// Restart after complete run
IF NOT Start_old AND Start THEN
	Index := 0;
	Finished := FALSE;
END_IF


CASE Index OF	
	0: // Switch to state 'Switch on disabled'
		IF (Start) THEN
			Mode_of_operation := E_Mode_of_operation.No_mode_active;
			Controlword := CONTROLWORD_STATE_CHANGE(Current_State, E_Statemachine_State.Switch_on_disabled);
			IF (Current_State = E_Statemachine_State.Switch_on_disabled) THEN			
				Index := Index + 2;
			ELSE
				Index := Index + 1;		
			END_IF
		END_IF
		
			
	1: // Wait for 'Switch on disabled'
		Controlword := CONTROLWORD_STATE_CHANGE(Current_State, E_Statemachine_State.Switch_on_disabled);	
		IF (Current_State = E_Statemachine_State.Switch_on_disabled) THEN			
			Index := Index + 1;		
		END_IF
					
		
	2: // Set Mode of operation
		Mode_of_operation := E_Mode_of_operation.Homing_mode;	
		Controlword := CONTROLWORD_STATE_CHANGE(Current_State, E_Statemachine_State.Switch_on_disabled);				
		IF (PDO.Mode_of_operation_display = E_Mode_of_operation.Homing_mode) THEN			
			IF Homing_parameters.Homing_mode = E_Homing_mode.Homing_on_current_position THEN
				Index := Index + 1 + 3*2;
			ELSE
				Index := Index + 1;		
			END_IF
		END_IF

		
	3: // Set Speed during search for switch		
		Controlword := CONTROLWORD_STATE_CHANGE(Current_State, E_Statemachine_State.Switch_on_disabled);	
		WriteData[0] := DWORD_TO_BYTE(Homing_parameters.Speed_switch);
		WriteData[1] := DWORD_TO_BYTE(SHR(Homing_parameters.Speed_switch,8));
		WriteData[2] := DWORD_TO_BYTE(SHR(Homing_parameters.Speed_switch,16));
		WriteData[3] := DWORD_TO_BYTE(SHR(Homing_parameters.Speed_switch,24));	
		SDO_WRITE(	
			AdsNetID		:= GLB.ADSNetID_CAN,
			PortNr			:= 16#1000 + GLB.NodeID,
			CO_Index		:= 16#6099,
			CO_SubIndex		:= 16#01,
			DataLength		:= 4,
			WriteData		:= WriteData,
			StartWriting	:= TRUE	
		);	
		Index := Index + 1;		
		
	4: // Wait for finish sdo transfer	
		Controlword := CONTROLWORD_STATE_CHANGE(Current_State, E_Statemachine_State.Switch_on_disabled);	
		SDO_WRITE(StartWriting := FALSE);
		IF SDO_WRITE.WriteDataFinished THEN
			Index := Index + 1;			
		END_IF	
		
		
	5: // Set Spped during search for zero			
		Controlword := CONTROLWORD_STATE_CHANGE(Current_State, E_Statemachine_State.Switch_on_disabled);	
		WriteData[0] := DWORD_TO_BYTE(Homing_parameters.Speed_zero);
		WriteData[1] := DWORD_TO_BYTE(SHR(Homing_parameters.Speed_zero,8));
		WriteData[2] := DWORD_TO_BYTE(SHR(Homing_parameters.Speed_zero,16));
		WriteData[3] := DWORD_TO_BYTE(SHR(Homing_parameters.Speed_zero,24));	
		SDO_WRITE(	
			AdsNetID		:= GLB.ADSNetID_CAN,
			PortNr			:= 16#1000 + GLB.NodeID,
			CO_Index		:= 16#6099,
			CO_SubIndex		:= 16#02,
			DataLength		:= 4,
			WriteData		:= WriteData,
			StartWriting	:= TRUE	
		);	
		Index := Index + 1;		
		
	6: // Wait for finish sdo transfer	
		Controlword := CONTROLWORD_STATE_CHANGE(Current_State, E_Statemachine_State.Switch_on_disabled);	
		SDO_WRITE(StartWriting := FALSE);
		IF SDO_WRITE.WriteDataFinished THEN
			Index := Index + 1;			
		END_IF		
		
		
	7: // Set Homing acceleration		
		Controlword := CONTROLWORD_STATE_CHANGE(Current_State, E_Statemachine_State.Switch_on_disabled);	
		WriteData[0] := DWORD_TO_BYTE(Homing_parameters.Acceleration);
		WriteData[1] := DWORD_TO_BYTE(SHR(Homing_parameters.Acceleration,8));
		WriteData[2] := DWORD_TO_BYTE(SHR(Homing_parameters.Acceleration,16));
		WriteData[3] := DWORD_TO_BYTE(SHR(Homing_parameters.Acceleration,24));	
		SDO_WRITE(	
			AdsNetID		:= GLB.ADSNetID_CAN,
			PortNr			:= 16#1000 + GLB.NodeID,
			CO_Index		:= 16#609A,
			CO_SubIndex		:= 16#00,
			DataLength		:= 4,
			WriteData		:= WriteData,
			StartWriting	:= TRUE	
		);	
		Index := Index + 1;		
		
	8: // Wait for finish sdo transfer	
		Controlword := CONTROLWORD_STATE_CHANGE(Current_State, E_Statemachine_State.Switch_on_disabled);	
		SDO_WRITE(StartWriting := FALSE);
		IF SDO_WRITE.WriteDataFinished THEN
			Index := Index + 1;			
		END_IF	
		
		
	9: // Set Homing mode		
		Controlword := CONTROLWORD_STATE_CHANGE(Current_State, E_Statemachine_State.Switch_on_disabled);	
		WriteData[0] := Homing_parameters.Homing_mode;
		SDO_WRITE(	
			AdsNetID		:= GLB.ADSNetID_CAN,
			PortNr			:= 16#1000 + GLB.NodeID,
			CO_Index		:= 16#6098,
			CO_SubIndex		:= 16#00,
			DataLength		:= 1,
			WriteData		:= WriteData,
			StartWriting	:= TRUE	
		);	
		Index := Index + 1;		
		
	10: // Wait for finish sdo transfer	
		Controlword := CONTROLWORD_STATE_CHANGE(Current_State, E_Statemachine_State.Switch_on_disabled);	
		SDO_WRITE(StartWriting := FALSE);
		IF SDO_WRITE.WriteDataFinished THEN
			Index := Index + 1;			
		END_IF		
		
		
	11: // Switch State to 'Operation enabled'
		Controlword := CONTROLWORD_STATE_CHANGE(Current_State, E_Statemachine_State.Operation_enabled);		
		IF (Current_State = E_Statemachine_State.Operation_enabled) THEN			
			Index := Index + 1;
		END_IF
		
		
	12: // Start homing and wait for finish
		Controlword := 16#1F;		
		IF (Statusword AND E_Statusword_Bits.HM_Homing_attained) <> 0 THEN			
			Index := Index + 1;		
		END_IF
	
		
	13: // Switch State to 'Switch on disabled'
		Controlword := CONTROLWORD_STATE_CHANGE(Current_State, E_Statemachine_State.Switch_on_disabled);	
		IF Current_State = E_Statemachine_State.Switch_on_disabled THEN			
			Index := 255;
		END_IF
		
		
	255: // Finished 
		Controlword := CONTROLWORD_STATE_CHANGE(Current_State, E_Statemachine_State.Switch_on_disabled);	
		FINISHED := TRUE;
				
		
	ELSE
		Index := 255;
			
END_CASE


Start_old := Start;

END_FUNCTION_BLOCK

// ---- POUs/FB/FB_Sequenz_Testing.TcPOU
FUNCTION_BLOCK FB_Sequenz_Testing
VAR_INPUT	
	Start			: BOOL 			:= FALSE;			// Start command
	Sequence_Name	: STRING(50) 	:= '';				// The name of the sequence
	Logging_active	: BOOL 			:= TRUE;			// The logging is default active. For deactivating set the variable to false.
END_VAR
VAR_OUTPUT
	Busy			: BOOL			:= FALSE;
	Finished		: BOOL			:= FALSE;			// The sequence is finished.
	Error			: BOOL			:= FALSE;			// Error during the sequence.
END_VAR
VAR_IN_OUT
	Step_list		: ARRAY [*] OF E_Test_step;	// Array with the sequence of steps
END_VAR
VAR
	Step_index		: DINT			:= 0;				// The current index of test step
	Step_state		: BYTE			:= 0;				// The internal state of the current test step
	Counter			: WORD			:= 0;				// Counter variable for internal use
	
	Name			: STRING(50)	:= '';				// The current sequence name. The name is saved once by start of the sequence.
	
	Data			: ARRAY [0..255] OF BYTE;
	CAN_Object		: ST_CAN_Object;	
	SDO_READ		: FB_SDO_READ;
	SDO_WRITE		: FB_SDO_WRITE;
	Write_busy		: BOOL 			:= FALSE;			// A writing process is running. After finishing the process the next test step is started
	Write_sequence	: BOOL			:= FALSE;			// If this Flag is set, the internal step state is increased. Otherwise the test step is finished after the write process.
	
	Next_Step_state	: BOOL 			:= FALSE;			// Increase the internal state of the test step
	Step_Finished	: BOOL 			:= FALSE;			// Switch to the next test step
	Error_step		: DINT 			:= -1;				// List index of the test state, at which an error is occured
	
	Current_Statemachine_state: E_Statemachine_State;	// The current State machine state
	
	Timeout_Counter	: INT			:= 0;				// Timeout Counter
	Timeout_Max		: INT			:= 0;				// Value at which the timeout counter is triggered (x 10 ms)

	Wait_Counter	: INT			:= 0;				// Wait Counter
	Wait_Step_Finish: BOOL			:= TRUE;			// True: The step is finished after the waiting time. False: The status counter in the step is increased after the waiting time.
	Wait_Time		: INT			:= 0;				// Value at which the wait counter is triggered (x 10 ms)

	Message			: STRING(60)	:= '';				// This message is send at the end of the FB
END_VAR

// Start / Reset
IF Start AND NOT Busy THEN
	Step_index		:= 0;
	Step_state 		:= 0;	
	Finished		:= FALSE;
	Error			:= FALSE;
	Error_step		:= -1;
 	Busy 			:= TRUE;	
	Name 			:= Sequence_Name;
	IF Sequence_Name = '' AND Logging_active THEN
		GLB.Logger(Message:='Start sequence');
	ELSE
		GLB.Logger(Message:=CONCAT('Start sequence: ', Sequence_Name)); 
	END_IF
END_IF


IF Busy THEN
	// Reached end?
	IF (Step_index > UPPER_BOUND(Step_list, 1)) OR (Error_step > -1) THEN
		Busy 		:= FALSE;
		Finished 	:= TRUE;
		IF Error_step = -1 AND Logging_active THEN
			GLB.Logger(Message:='Sequence successful', SaveFlag:=TRUE);
			Error	:= FALSE;
		ELSE	
			GLB.Logger(Message:='Sequence failed', SaveFlag:=TRUE);			
			Error	:= TRUE;		
		END_IF
				
	ELSE
		// Get the current state of the State machine
		Current_Statemachine_state 			:= GET_STATE(PDO.Statusword);
			
		// Processing the individual test steps  
		CASE Step_list[Step_index] OF
		
			// **** Change of state machine state *****
			// Switch directly to state 'Switch on disabled' -> Set Controlword to 0
			E_Test_step.Switch_on_disabled:
				CASE Step_state OF
					0:	// Set Controlword to 0
						PDO.Controlword			:= E_Statemachine_Transition_Controlword.Switch_on_disabled;
						Message					:= 'Switch to state Switch on disabled';		
						Next_Step_state			:= TRUE;
					
					1:	// Wait until state 'Switch on disabled'
						IF Current_Statemachine_state = E_Statemachine_State.Switch_on_disabled THEN		Step_Finished := TRUE;	END_IF	
				END_CASE	
				
			// Switch directly to state 'Quick stop active' -> Set Controlword to 2		
			E_Test_step.Quick_stop_active:
				CASE Step_state OF
					0:	// Set Controlword to 2
						PDO.Controlword			:= E_Statemachine_Transition_Controlword.Quick_stop_active;
						Message					:= 'Switch to state Quick stop active';		
						Next_Step_state			:= TRUE;
					
					1:	// Wait until state 'Quick stop active'
						IF Current_Statemachine_state = E_Statemachine_State.Quick_stop_active THEN			Step_Finished := TRUE;	END_IF
				END_CASE
													
			// Switch directly to state 'Ready to switch on' -> Set Controlword to 6		
			E_Test_step.Ready_to_switch_on:
				CASE Step_state OF
					0:	// Set Controlword to 6
						PDO.Controlword			:= E_Statemachine_Transition_Controlword.Ready_to_switch_on;
						Message					:= 'Switch to state Ready to switch on';			
						Next_Step_state			:= TRUE;				
				
					1:	// Wait until state 'Ready to switch on'
						IF Current_Statemachine_state = E_Statemachine_State.Ready_to_switch_on THEN		Step_Finished := TRUE;	END_IF
				END_CASE
													
			// Switch directly to state 'Switched on' -> Set Controlword to 7			
			E_Test_step.Switched_on:				
				CASE Step_state OF
					0:	// Set Controlword to 7
						PDO.Controlword			:= E_Statemachine_Transition_Controlword.Switched_on;
						Message					:= 'Switch to state Switched on';				
						Next_Step_state			:= TRUE;
					
					1:	// Wait until state 'Switched on'
						IF Current_Statemachine_state = E_Statemachine_State.Switched_on THEN				Step_Finished := TRUE;	END_IF
				END_CASE
													
			// Switch directly to state 'Operation enabled' -> Set Controlword to F		
			E_Test_step.Operation_enabled:				
				CASE Step_state OF
					0:	// Set Controlword to F
						PDO.Controlword			:= E_Statemachine_Transition_Controlword.Operation_enabled;
						Message					:= 'Switch to state Operation enabled';			
						Next_Step_state			:= TRUE;
					
					1:	// Wait until state 'Operation enabled'
						IF Current_Statemachine_state = E_Statemachine_State.Operation_enabled THEN			Step_Finished := TRUE;	END_IF
				END_CASE													
			// ****************************************	
						
			// ***** Change of Mode of Operation ******
			// Set Mode of Operation to 'No mode'
			E_Test_step.No_Mode:
				CASE Step_state OF
					0:
						PDO.Mode_of_operation	:= E_Mode_of_Operation.No_mode_active;
						Message					:= 'Set Mode of Operation to "No mode"';		
						Next_Step_state			:= TRUE;
					
					1:	// Wait until mode 'No mode'
						IF PDO.Mode_of_operation_display = E_Mode_of_Operation.No_mode_active THEN			Step_Finished := TRUE;	END_IF				
				END_CASE
						
			// Set Mode of Operation to 'Profile Position Mode'
			E_Test_step.Mode_PPM:
				CASE Step_state OF
					0:	
						PDO.Mode_of_operation	:= E_Mode_of_Operation.Profile_position_mode;
						Message					:= 'Set Mode of Operation to "Profile Position Mode"';			
						Next_Step_state			:= TRUE;
					
					1:	// Wait until mode 'Profile Position Mode'
						IF PDO.Mode_of_operation_display = E_Mode_of_Operation.Profile_position_mode THEN	Step_Finished := TRUE;	END_IF				
				END_CASE
								
			// Set Mode of Operation to 'Velocity Mode'
			E_Test_step.Mode_VM:
				CASE Step_state OF
					0:
						PDO.Mode_of_operation	:= E_Mode_of_Operation.Velocity_mode;
						Message					:= 'Set Mode of Operation to "Velocity Mode"';			
						Next_Step_state			:= TRUE;
					
					1:	// Wait until mode 'Velocity Mode'
						IF PDO.Mode_of_operation_display = E_Mode_of_Operation.Velocity_mode THEN			Step_Finished := TRUE;	END_IF		
				END_CASE
			
			// Set Mode of Operation to 'Profile Velocity Mode'
			E_Test_step.Mode_PVM:
				CASE Step_state OF
					0:
						PDO.Mode_of_operation	:= E_Mode_of_Operation.Profile_velocity_mode;
						Message					:= 'Set Mode of Operation to "Profile Velocity Mode"';			
						Next_Step_state			:= TRUE;
					
					1:	// Wait until mode 'Profile Velocity Mode'
						IF PDO.Mode_of_operation_display = E_Mode_of_Operation.Profile_velocity_mode THEN	Step_Finished := TRUE;	END_IF		
				END_CASE
										
			// Set Mode of Operation to 'Profile Torque Mode'
			E_Test_step.Mode_PTM:
				CASE Step_state OF
					0:
						PDO.Mode_of_operation	:= E_Mode_of_Operation.Profile_torque_mode;
						Message					:= 'Set Mode of Operation to "Profile Torque Mode"';		
						Next_Step_state			:= TRUE;
					
					1:	// Wait until mode 'Profile Torque Mode'
						IF PDO.Mode_of_operation_display = E_Mode_of_Operation.Profile_torque_mode THEN		Step_Finished := TRUE;	END_IF		
				END_CASE
				
			// Set Mode of Operation to 'Homing Mode'
			E_Test_step.Mode_HM:
				CASE Step_state OF
					0:
						PDO.Mode_of_operation	:= E_Mode_of_Operation.Homing_mode;
						Message					:= 'Set Mode of Operation to "Homing mode"';
						Next_Step_state			:= TRUE;
					
					1:	// Wait until mode 'Homing Mode'
						IF PDO.Mode_of_operation_display = E_Mode_of_Operation.Homing_mode THEN				Step_Finished := TRUE;	END_IF		
				END_CASE
										
			// Set Mode of Operation to 'Interpolated Position Mode'
			E_Test_step.Mode_IPM:
				CASE Step_state OF
					0:
						PDO.Mode_of_operation	:= E_Mode_of_Operation.Interpolated_position_mode;
						Message					:= 'Set Mode of Operation to "Interpolated Position Mode"';
						Next_Step_state			:= TRUE;
					
					1:	// Wait until mode 'Interpolated Position Mode'
						IF PDO.Mode_of_operation_display = E_Mode_of_Operation.Interpolated_position_mode THEN	Step_Finished := TRUE;	END_IF		
				END_CASE
			// ****************************************	
						
			// ************** Init steps **************	
			// Set the factor group to use rpm as user-defined velocity unit
			E_Test_step.Factor_group_rpm:
				Write_busy := TRUE;
				CASE Step_state OF
					0:	// Set ...
						Write_sequence := TRUE;
						DWORD_TO_BYTE_ARRAY(4096, Data);			
						CAN_Object 		:= DS402_Object_List.Velocity_Factor_Numerator;
						
					2:	// Set ...
						Write_sequence := FALSE;					
						DWORD_TO_BYTE_ARRAY(60, Data);			
						CAN_Object 		:= DS402_Object_List.Velocity_Factor_Divisor;
						
						
						
				END_CASE	
			// ****************************************	
			
			// ************ Setting values ************	
			// Set 'Velocity_window' to value 30
			E_Test_step.Velocity_window_30rpm:
				CASE Step_state OF
					0:
						DWORD_TO_BYTE_ARRAY(30, Data);			
						CAN_Object 		:= DS402_Object_List.Velocity_window;
						Message 		:= 'Set Velocity_window to 30';					
						Write_busy		:= TRUE;		
				END_CASE
			
			// Set 'Velocity window time' to value 100
			E_Test_step.Velocity_window_100ms:
				CASE Step_state OF
					0:
						DWORD_TO_BYTE_ARRAY(100, Data);			
						CAN_Object 		:= DS402_Object_List.Velocity_window_time;
						Message			:= 'Set Velocity window time to 100';					
						Write_busy		:= TRUE;
				END_CASE
				
			// Set 'Profile acceleration' to value 1000
			E_Test_step.Acceleration_1000:
				CASE Step_state OF
					0:
						DWORD_TO_BYTE_ARRAY(1000, Data);			
						CAN_Object 		:= DS402_Object_List.Profile_acceleration;
						Message			:= 'Set Profile acceleration to 1000';
						Write_busy		:= TRUE;	
				END_CASE
				
			// Set 'Profile deceleration' to value 1000			
			E_Test_step.Deceleration_1000:
				CASE Step_state OF
					0:
						DWORD_TO_BYTE_ARRAY(1000, Data);	
						CAN_Object 		:= DS402_Object_List.Profile_deceleration; 				
						Message			:= 'Set Profile deceleration to 1000';
						Write_busy		:= TRUE;
				END_CASE
				
			// Set 'Profile velocity' to value 1000			
			E_Test_step.PPM_Velocity_1000:
				CASE Step_state OF
					0:
						DWORD_TO_BYTE_ARRAY(1000, Data);			
						CAN_Object 		:= DS402_Object_List.Profile_velocity;
						Message			:= 'Set Profile velocity to 1000';					
						Write_busy		:= TRUE;	
				END_CASE
	
			// Set 'Target velocity' to value 1000
			E_Test_step.PVM_Velocity_1000:
				CASE Step_state OF
					0:	
						DWORD_TO_BYTE_ARRAY(1000, Data);			
						CAN_Object 		:= DS402_Object_List.Target_velocity;
						Message			:= 'Set Target velocity to 1000';
						Write_busy		:= TRUE;
				END_CASE		
			// ****************************************	
							
			// *********** Check conditions ***********
			// Check if the 'Target reached' bit in statusword is set within 200 ms
			E_Test_step.Check_Statusword_Target_reached_200ms:
				Timeout_Max 		:= 20;
				IF (PDO.Statusword AND E_Statusword_Bits.Target_reached) = E_Statusword_Bits.Target_reached THEN
					Message			:= 'Target reached bit is set';
					Step_Finished	:= TRUE;					
				END_IF	
			// ****************************************				
			
			// ************ Waiting times *************
			E_Test_step.Wait_10ms:		IF Step_state = 0 THEN	Wait_Time := 1; 	Message := 'Wait Time 10 ms is running';	Next_Step_State:=TRUE; END_IF
			E_Test_step.Wait_50ms:		IF Step_state = 0 THEN	Wait_Time := 5; 	Message := 'Wait Time 50 ms is running';	Next_Step_State:=TRUE; END_IF
			E_Test_step.Wait_100ms:		IF Step_state = 0 THEN	Wait_Time := 10; 	Message := 'Wait Time 100 ms is running';	Next_Step_State:=TRUE; END_IF
			E_Test_step.Wait_250ms:		IF Step_state = 0 THEN	Wait_Time := 25; 	Message := 'Wait Time 250 ms is running';	Next_Step_State:=TRUE; END_IF
			E_Test_step.Wait_500ms:		IF Step_state = 0 THEN	Wait_Time := 50; 	Message := 'Wait Time 500 ms is running';	Next_Step_State:=TRUE; END_IF
			E_Test_step.Wait_1000ms:	IF Step_state = 0 THEN	Wait_Time := 100; 	Message := 'Wait Time 1 s is running';		Next_Step_State:=TRUE; END_IF
			E_Test_step.Wait_2500ms:	IF Step_state = 0 THEN	Wait_Time := 250; 	Message := 'Wait Time 2.5 s is running';	Next_Step_State:=TRUE; END_IF
			// Feel free to create your own needed wait times :-)
			// ****************************************		
						
			ELSE
				// unknown steps -> next step
				Message				:= CONCAT(CONCAT('FB_Start_Testing: ERROR, unknown test step (', DINT_TO_STRING(Step_index)), ')');
				Step_Finished		:= TRUE;
	
		END_CASE
		
		// Waiting time. Active, if Wait_Time is greater than 0
		IF Wait_Time > 0 THEN
			Wait_Counter			:= Wait_Counter + 1;	
			IF Wait_Counter >= Wait_Time THEN
				Message				:= 'Waiting time expired';			
				IF Wait_Step_Finish THEN 
					Step_Finished	:= TRUE;
				ELSE
					Next_Step_state	:= TRUE;
				END_IF
			END_IF
		END_IF
		
		// SDO Write process is running. This generell function is used, if Write_busy is set.
		IF Write_busy THEN
			IF Step_state.0 = 0 THEN
				// Start writing
				SDO_Write(
					ADSNetID		:= GLB.ADSNetID_CAN,				
					PortNr 		 	:= 16#1000 + GLB.NodeID,
					CO_Index 		:= CAN_Object.Index,
					CO_SubIndex 	:= CAN_Object.Subindex,
					DataLength 		:= CAN_Object.Length,
					WriteData		:= Data,
					StartWriting	:= TRUE	);
				Next_Step_state	:= TRUE;								
			ELSE
				// Wait for finishing
				SDO_Write(StartWriting:=FALSE);
				IF SDO_WRITE.WriteDataFinished THEN
					Write_busy			:= FALSE;
					IF SDO_WRITE.Error = 0 THEN									
						IF Write_sequence THEN
							Next_step_state	:= TRUE;
						ELSE						
							Step_Finished	:= TRUE;
						END_IF;
					ELSE
						Message			:= CONCAT('ERROR: Write failed, Errornumber: ', DWORD_TO_HEXSTR(SDO_WRITE.Error, 8, FALSE));
						Error_step		:= Step_index;		
					END_IF	
					SDO_Write();	
				END_IF
			END_IF
		END_IF
		
		// Next Test step
		IF Step_Finished THEN
			IF Message = '' THEN Message := 'OK'; END_IF
			Step_Finished 			:= FALSE;
			Step_index				:= Step_index + 1;
			Step_state 				:= 0;
			Wait_Counter			:= 0;
			Wait_Time				:= 0;
			Wait_Step_Finish		:= TRUE;
			Write_sequence			:= FALSE;
			Timeout_Counter			:= 0;
			Timeout_Max 			:= 10;			// Set Timeout to a default value of 10 (= 100 ms)
			
		// Next internal state of the test step			
		ELSIF Next_Step_state THEN
			Next_Step_state			:= FALSE;
			Step_state				:= Step_state + 1;
			Timeout_Counter			:= 0;	
		
		// Timeout
		ELSE
			IF Timeout_Max > 0 THEN
				IF Timeout_Counter >= Timeout_Max THEN
					Message			:= CONCAT(CONCAT('Timeout triggered (', INT_TO_STRING(Timeout_Max * 10)), ' ms)');
					Error_step		:= Step_index;
				END_IF
				Timeout_Counter	:= Timeout_Counter + 1;	
			END_IF
		END_IF
	END_IF
	
	
	// Log message
	IF Message <> '' AND Logging_active  THEN
		GLB.Logger(Message:=Message);
		Message := '';
	END_IF
END_IF

END_FUNCTION_BLOCK

// ---- POUs/GET_STATE.TcPOU
FUNCTION GET_STATE : E_Statemachine_State
VAR_INPUT
	Statusword: WORD;
END_VAR
VAR_OUTPUT
	State : E_Statemachine_State;
END_VAR
VAR_STAT
	State_State: ARRAY[0..7] OF E_Statemachine_State := [
		E_Statemachine_State.Not_ready_to_switch_on,
		E_Statemachine_State.Switch_on_disabled,
		E_Statemachine_State.Ready_to_switch_on,
		E_Statemachine_State.Switched_on,
		E_Statemachine_State.Operation_enabled,
		E_Statemachine_State.Quick_stop_active,
		E_Statemachine_State.Fault_reaction_active,
		E_Statemachine_State.Fault];
			
	State_Statusword: ARRAY[0..7] OF WORD := [ 
		16#00,	// Not ready to switch on
		16#40, 	// Switch on disabled
		16#21, 	// Ready to switch on
		16#23, 	// Switched on
		16#27, 	// Operation enable
		16#07, 	// Quick_stop_active
		16#0F,	// Fault_reaction_active
		16#08];	// Fault
		
	State_Mask: ARRAY[0..7] OF WORD := [ 
		16#4F,	// Not ready to switch on
		16#4F, 	// Switch on disabled
		16#6F, 	// Ready to switch on
		16#6F, 	// Switched on
		16#6F, 	// Operation enable
		16#6F, 	// Quick_stop_active
		16#4F,	// Fault_reaction_active
		16#4F];	// Fault	
END_VAR
VAR
	i: INT;
END_VAR

FOR i := 0 TO 7 DO
	IF (Statusword AND State_Mask[i]) = State_Statusword[i] THEN
		State 		:= State_State[i];
		GET_STATE 	:= State_State[i];
		EXIT;
	END_IF
END_FOR

END_FUNCTION

// ---- POUs/Velocity_Mode.TcPOU
FUNCTION_BLOCK Velocity_Mode
VAR_INPUT
	NodeID			: BYTE; (* This Port No. addresses the CANopen Node (see System Manager) *)
	Start 			: BOOL;
	Current_State 	: E_Statemachine_State;	
	Statusword		: WORD;	
	Velocity_parameters	: ST_Velocity_parameters;
END_VAR
VAR_OUTPUT
	Controlword 	: WORD;
	Mode_of_operation 	: E_Mode_of_operation	:= E_Mode_of_operation.No_mode_active;
	vl_target_velocity	: INT := 0;	
	Finished		: BOOL;
END_VAR
VAR
	Index 			: BYTE := 0;
	
	SDO_WRITE		: FB_SDO_WRITE;
	WriteData		: ARRAY [0..255] OF BYTE;
	
	SDO_READ		: FB_SDO_READ;
	ReadStart		: BOOL;
	ReadError		: DWORD;
	ReadData		: ARRAY [0..255] OF BYTE;
	
	fbTonDelay		: TON;
	Start_old		: BOOL := FALSE;
END_VAR

// Restart after complete run
IF NOT Start_old AND Start THEN
	Index := 0;
	Finished := FALSE;
END_IF


CASE Index OF	
	0: // Switch to state 'Switch on disabled'
		IF (Start) THEN
			Mode_of_operation := E_Mode_of_operation.No_mode_active;
			vl_target_velocity := 0;			
			Controlword := CONTROLWORD_STATE_CHANGE(Current_State, E_Statemachine_State.Switch_on_disabled);
			IF (Current_State = E_Statemachine_State.Switch_on_disabled) THEN			
				Index := Index + 2;
			ELSE
				Index := Index + 1;		
			END_IF
		END_IF
		
			
	1: // Wait for 'Switch on disabled'
		Controlword := CONTROLWORD_STATE_CHANGE(Current_State, E_Statemachine_State.Switch_on_disabled);	
		IF (Current_State = E_Statemachine_State.Switch_on_disabled) THEN			
			Index := Index + 1;		
		END_IF
					
		
	2: // Set Mode of operation and Acceleration
		Mode_of_operation := E_Mode_of_operation.Velocity_mode;	
		Controlword := CONTROLWORD_STATE_CHANGE(Current_State, E_Statemachine_State.Switch_on_disabled);				
		WriteData[0] := DWORD_TO_BYTE(Velocity_parameters.vl_velocity_acceleration);
		WriteData[1] := DWORD_TO_BYTE(SHR(Velocity_parameters.vl_velocity_acceleration,8));
		WriteData[2] := DWORD_TO_BYTE(SHR(Velocity_parameters.vl_velocity_acceleration,16));
		WriteData[3] := DWORD_TO_BYTE(SHR(Velocity_parameters.vl_velocity_acceleration,24));	
		SDO_WRITE(	
			AdsNetID		:= GLB.ADSNetID_CAN,
			PortNr			:= 16#1000 + GLB.NodeID,
			CO_Index		:= 16#6048,
			CO_SubIndex		:= 16#00,
			DataLength		:= 4,
			WriteData		:= WriteData,
			StartWriting	:= TRUE	
		);	
		Index := Index + 1;		
		
	3: // Wait for finish sdo transfer	
		Controlword := CONTROLWORD_STATE_CHANGE(Current_State, E_Statemachine_State.Switch_on_disabled);	
		SDO_WRITE(StartWriting := FALSE);
		IF SDO_WRITE.WriteDataFinished THEN
			Index := Index + 1;			
		END_IF	
		
		
	4: // Set Deceleration			
		Controlword := CONTROLWORD_STATE_CHANGE(Current_State, E_Statemachine_State.Switch_on_disabled);	
		WriteData[0] := DWORD_TO_BYTE(Velocity_parameters.vl_velocity_deceleration);
		WriteData[1] := DWORD_TO_BYTE(SHR(Velocity_parameters.vl_velocity_deceleration,8));
		WriteData[2] := DWORD_TO_BYTE(SHR(Velocity_parameters.vl_velocity_deceleration,16));
		WriteData[3] := DWORD_TO_BYTE(SHR(Velocity_parameters.vl_velocity_deceleration,24));	
		SDO_WRITE(	
			AdsNetID		:= GLB.ADSNetID_CAN,
			PortNr			:= 16#1000 + GLB.NodeID,
			CO_Index		:= 16#6049,
			CO_SubIndex		:= 16#00,
			DataLength		:= 4,
			WriteData		:= WriteData,
			StartWriting	:= TRUE	
		);	
		Index := Index + 1;		
		
	5: // Wait for finish sdo transfer	
		Controlword := CONTROLWORD_STATE_CHANGE(Current_State, E_Statemachine_State.Switch_on_disabled);	
		SDO_WRITE(StartWriting := FALSE);
		IF SDO_WRITE.WriteDataFinished THEN
			Index := Index + 1;			
		END_IF		
		
		
	6: // Set Velocity and switch State to 'Operation enabled'
		vl_target_velocity := Velocity_parameters.vl_target_velocity;
		Controlword := CONTROLWORD_STATE_CHANGE(Current_State, E_Statemachine_State.Operation_enabled);		
		IF (Current_State = E_Statemachine_State.Operation_enabled) THEN			
			Index := 255;
		END_IF
				
		
	255: // Finished 
		Controlword := CONTROLWORD_STATE_CHANGE(Current_State, E_Statemachine_State.Switch_on_disabled);	
		FINISHED := TRUE;
				
		
	ELSE
		Index := 255;
			
END_CASE


Start_old := Start;

END_FUNCTION_BLOCK

// ---- POUs/Profile_Velocity_Mode.TcPOU
FUNCTION_BLOCK Profile_Velocity_Mode
VAR_INPUT
	NodeID					: BYTE; (* This Port No. addresses the CANopen Node (see System Manager) *)
	Start 					: BOOL;
	Current_State 			: E_Statemachine_State;	
	Statusword				: WORD;	
	Profile_velocity_parameters	: ST_Profile_velocity_parameters;
END_VAR
VAR_OUTPUT
	Controlword 			: WORD;
	Mode_of_operation 		: E_Mode_of_operation	:= E_Mode_of_operation.No_mode_active;
	Target_velocity			: DINT;
	Encoder_offset			: WORD;
	Finished				: BOOL;
END_VAR
VAR
	Index 			: BYTE := 0;
	
	SDO_WRITE		: FB_SDO_WRITE;
	WriteData		: ARRAY [0..255] OF BYTE;
	
	Start_old		: BOOL := FALSE;
END_VAR

// Restart after complete run
IF NOT Start_old AND Start THEN
	Index := 0;
	Finished := FALSE;
END_IF


CASE Index OF	
	0: // Switch to state 'Switch on disabled'
		IF (Start) THEN
			Mode_of_operation := E_Mode_of_operation.No_mode_active;
			Target_velocity	:= 0;	
			Controlword := CONTROLWORD_STATE_CHANGE(Current_State, E_Statemachine_State.Switch_on_disabled);
			IF (Current_State = E_Statemachine_State.Switch_on_disabled) THEN			
				Index := Index + 2;
			ELSE
				Index := Index + 1;		
			END_IF
		END_IF
		
			
	1: // Wait for 'Switch on disabled'
		Controlword := CONTROLWORD_STATE_CHANGE(Current_State, E_Statemachine_State.Switch_on_disabled);	
		IF (Current_State = E_Statemachine_State.Switch_on_disabled) THEN			
			Index := Index + 1;		
		END_IF
		
		
	2: // Set Mode of operation and Acceleration
		Mode_of_operation := E_Mode_of_operation.Profile_velocity_mode;	
		Controlword := CONTROLWORD_STATE_CHANGE(Current_State, E_Statemachine_State.Switch_on_disabled);				
		WriteData[0] := DWORD_TO_BYTE(Profile_velocity_parameters.Profile_acceleration);
		WriteData[1] := DWORD_TO_BYTE(SHR(Profile_velocity_parameters.Profile_acceleration,8));
		WriteData[2] := DWORD_TO_BYTE(SHR(Profile_velocity_parameters.Profile_acceleration,16));
		WriteData[3] := DWORD_TO_BYTE(SHR(Profile_velocity_parameters.Profile_acceleration,24));	
		SDO_WRITE(	
			AdsNetID		:= GLB.ADSNetID_CAN,
			PortNr			:= 16#1000 + GLB.NodeID,
			CO_Index		:= 16#6083,
			CO_SubIndex		:= 16#00,
			DataLength		:= 4,
			WriteData		:= WriteData,
			StartWriting	:= TRUE	
		);	
		Index := Index + 1;		
		
	3: // Wait for finish sdo transfer	
		Controlword := CONTROLWORD_STATE_CHANGE(Current_State, E_Statemachine_State.Switch_on_disabled);	
		SDO_WRITE(StartWriting := FALSE);
		IF SDO_WRITE.WriteDataFinished THEN
			Index := Index + 1;			
		END_IF	
		
		
	4: // Set Deceleration			
		Controlword := CONTROLWORD_STATE_CHANGE(Current_State, E_Statemachine_State.Switch_on_disabled);	
		WriteData[0] := DWORD_TO_BYTE(Profile_velocity_parameters.Profile_deceleration);
		WriteData[1] := DWORD_TO_BYTE(SHR(Profile_velocity_parameters.Profile_deceleration,8));
		WriteData[2] := DWORD_TO_BYTE(SHR(Profile_velocity_parameters.Profile_deceleration,16));
		WriteData[3] := DWORD_TO_BYTE(SHR(Profile_velocity_parameters.Profile_deceleration,24));	
		SDO_WRITE(	
			AdsNetID		:= GLB.ADSNetID_CAN,
			PortNr			:= 16#1000 + GLB.NodeID,
			CO_Index		:= 16#6084,
			CO_SubIndex		:= 16#00,
			DataLength		:= 4,
			WriteData		:= WriteData,
			StartWriting	:= TRUE	
		);	
		Index := Index + 1;		
		
	5: // Wait for finish sdo transfer	
		Controlword := CONTROLWORD_STATE_CHANGE(Current_State, E_Statemachine_State.Switch_on_disabled);	
		SDO_WRITE(StartWriting := FALSE);
		IF SDO_WRITE.WriteDataFinished THEN
			Index := Index + 1;			
		END_IF					
		
	6: // Set  velocity	
		Controlword := CONTROLWORD_STATE_CHANGE(Current_State, E_Statemachine_State.Switch_on_disabled);	
		Target_velocity	:= Profile_velocity_parameters.Target_velocity;
		Index := Index + 1;		
		
	7: // Switch State to 'Operation enabled'
		Controlword := CONTROLWORD_STATE_CHANGE(Current_State, E_Statemachine_State.Operation_enabled);		
		IF (Current_State = E_Statemachine_State.Operation_enabled) THEN			
			Index := 255;
		END_IF
				
		
	255: // Finished 
		FINISHED := TRUE;
				
		
	ELSE
		Index := 255;
			
END_CASE


Start_old := Start;

END_FUNCTION_BLOCK

// ---- POUs/FUN/DWORD_TO_BYTE_ARRAY.TcPOU
FUNCTION DWORD_TO_BYTE_ARRAY
VAR_INPUT
	Value	: DWORD;
END_VAR
VAR_IN_OUT
	DATA	: ARRAY [*] OF BYTE;
END_VAR
VAR
	i		: BYTE := 0;
END_VAR

FOR i := 0 TO 3 DO
	DATA[i] := DWORD_TO_BYTE(SHR(Value, (8*i)));			
END_FOR;

END_FUNCTION

// ---- POUs/J_Stop_Testing_SM.TcPOU
FUNCTION_BLOCK J_Stop_Testing_SM
VAR_INPUT
	JST_NodeID					: BYTE; (* This Port No. addresses the CANopen Node (see System Manager) *)
	JST_Start_Testing			: BOOL; (* Send True to start the Stop Testing*)
	JST_Current_State 			: E_Statemachine_State;
END_VAR
VAR_OUTPUT
	Finished 					: BOOL := FALSE;
	JST_Controlword 			: WORD;
	Mode_of_operation 			: E_Mode_of_operation	:= E_Mode_of_operation.No_mode_active;
END_VAR
VAR
	// Statemachine variables
	e_Controlword_Send : (Wait_For_Send, Continue_SM) := Continue_SM;
	
	JST_Profile_Velocity_Mode 		: Profile_Velocity_Mode;
	e_Stop_Testing_State_Machine 	: (Idle,
									   Initialise_Drive,
									   Check_Start_Drive_Condition,
									   Change_Stop_Testing_State,
								       Stop_Testing, 
									   Check_Stop_Drive_Condition,
									   Start_Drive, 
									   Error_Handling); 
									
	e_Operation_Mode : E_Mode_of_operation := E_Mode_of_operation.Velocity_mode;
	
	(* e_Stop_Mode :  (Switch_On,					//schnell runterrampen -> Switched on
					Shutdown,					//Disable PS
					Switch_On_Disabled,			//Disable PS
					Vel_To_Zero,				//Ramp down
					Halt,						//stillstand mit dehmoment -> Weiterdrehen
					Quick_Stop,					//schnell runterrampen -> Switch on Disabled
					STO1,						//Disable PS
					STO2,						//Disable PS
					Fault						//DISABLE PS
					) := Switch_On; *)
	
	e_Stop_Mode : J_E_Stop_Modes := J_E_Stop_Modes.Switch_On;
	
	e_Stop_Type :  (Idle_Output_Stage,
				    Ramp_Down_AFAP,
					Vel_Zero);
					
	e_Start_Type : (Start_After_Reset,
					No_Start_After_Reset);
					
	
	JST_Profile_velocity_parameters	: ST_Profile_velocity_parameters := (Target_velocity 	  := 1000,
																 		 Profile_acceleration := 1000,
																 		 Profile_deceleration := 1000);
																 
	Target_velocity	: INT := 0;
	Target_State : E_STATEMACHINE_STATE;
	
	SDO_WRITE		: FB_SDO_WRITE;
	WriteData		: ARRAY [0..255] OF BYTE;
	
	//Tolerance variables
	Time_Tolerance : INT := 20;		//Unit is ms
	Vel_Tolerance  : INT := 30;		//Assumed that unit is RPM
	Stop_Tolerance : INT := 5;
	Stop_Time_AFAP : TIME := T#500MS;
	
	// Trash Variables 
	Temp 				         : BOOL := TRUE;
	JumpNextState 				 : BOOL := FALSE;
	Quick_Stop_Activ_Reset 		 : WORD := 16#00;
	Mode_Change 				 : BOOL := TRUE;
	Temp_msg 					 : STRING; 
	Delay 						 : BOOL := FALSE;
	Send_Controlword_Direct 	 : BOOL := FALSE;
	Quickstop_Change_Controlword : BOOL := TRUE;
	
	//Timer variables
	Toff : TIME := T#2000MS;
	
	StopTimer			 : TON := (PT := Toff);
	StartDelayTimer 	 : TON := (PT := Toff);
	CheckStartDelayTimer : TON := (PT := Toff);
	
	Stop_Timer 			: BOOL;
	Start_Delay_Timer 		: BOOL;
	Check_Start_Delay_Timer : BOOL;
	
	Elapsed_Time 			: TIME;
	
	//Message logging variables
	//fb_Message_Logging 		: J_Make_Message;
	Stop_Mode_String 		: STRING;
	
	// 24V Output variables
	OutputSTO1 	AT%Q* 		: BOOL;
	OutputSTO2 	AT%Q* 		: BOOL;

	Actual_Velocity_RPM		: DINT;
END_VAR

StopTimer(IN := Stop_Timer);
StartDelayTimer(IN := Start_Delay_Timer);
CheckStartDelayTimer(IN := Check_Start_Delay_Timer);

Actual_Velocity_RPM := PDO.vl_Velocity_actual_value;
//e_Operation_Mode := PDO.Mode_of_operation_display;

CASE e_Controlword_Send OF
	Continue_SM:		
		CASE e_Stop_Testing_State_Machine OF
			
			Idle:
				IF JST_Start_Testing THEN
					e_Stop_Testing_State_Machine := Initialise_Drive;
					e_Operation_Mode := E_Mode_of_operation.Velocity_mode;
					Finished := FALSE;
					GLB.Logger.OpenFlag := TRUE;
				ELSE
					e_Stop_Testing_State_Machine := Idle;
				END_IF
				
		//_____________________Start Drive SM___________________________________
			Initialise_Drive:
				OutputSTO1 := TRUE;
				OutputSTO2 := TRUE;
				CASE e_Operation_Mode OF
					//----------------------------------------------------------
					E_Mode_of_operation.Profile_position_mode:
						// Vel = 1000 ; Acc = 1000 ; Dec = 1000, Pos = 10000000						  
						IF NOT JST_Profile_Velocity_Mode.Finished THEN
							//just want to set acc and dec but not enable the drive
							JST_Profile_Velocity_Mode (NodeID := JST_NodeID,		//PVM just because the param for acc and dec are set and the same as in PPM
													   Start := TRUE,
													   Current_State := JST_Current_State,
													   Statusword := PDO.Statusword,
													   Profile_velocity_parameters := JST_Profile_velocity_parameters,
													   Controlword => JST_Controlword);
							e_Controlword_Send := Continue_SM;
							
						ELSIF JST_Profile_Velocity_Mode.Finished THEN

							PDO.Mode_of_operation 	:= E_Mode_of_operation.Profile_position_mode;		
							PDO.Profile_velocity 	:= JST_Profile_velocity_parameters.Target_velocity;
							PDO.Target_position 	:= 16#1000000;    // need to evaluate a good value 
							
							//Profile position FB how to use?
							Target_State := E_Statemachine_State.Operation_enabled;
							e_Controlword_Send := Wait_For_Send;
							e_Stop_Testing_State_Machine := Check_Start_Drive_Condition;
							Mode_Change := TRUE;
						END_IF
					//----------------------------------------------------------					
					E_Mode_of_operation.Velocity_mode:
							// Vel = 1000
							PDO.Mode_of_operation := E_Mode_of_Operation.Velocity_mode;
							PDO.vl_target_velocity := TO_INT(JST_Profile_velocity_parameters.Target_velocity);
							Target_State := E_Statemachine_State.Operation_enabled;
							e_Controlword_Send := Wait_For_Send;
							e_Stop_Testing_State_Machine := Check_Start_Drive_Condition;
							Check_Start_Delay_Timer := TRUE;	
		
					//----------------------------------------------------------	
					E_Mode_of_operation.Profile_velocity_mode:
						// Vel = 1000 ; Acc = 1000 ; Dec = 500
						// Start Drive, Wait for SDO written then change state
						IF NOT JST_Profile_Velocity_Mode.Finished THEN
							JST_Profile_Velocity_Mode (NodeID := JST_NodeID,
													   Start := TRUE,
													   Current_State := JST_Current_State,
													   Statusword := JST_Current_State,
													   Profile_velocity_parameters := JST_Profile_velocity_parameters,
													   Controlword => JST_Controlword);
							e_Controlword_Send := Continue_SM;
							
						ELSIF JST_Profile_Velocity_Mode.Finished THEN
							PDO.Profile_velocity := JST_Profile_velocity_parameters.Target_velocity;
							e_Stop_Testing_State_Machine := Check_Start_Drive_Condition;
						END_IF
					//----------------------------------------------------------
					E_Mode_of_operation.Profile_torque_mode:
						Target_State := E_Statemachine_State.Ready_to_switch_on;
						e_Controlword_Send := Wait_For_Send;
							IF PDO.Controlword = E_Statusword_Bits.Ready_to_switch_on THEN
								PDO.Mode_of_operation := E_Mode_of_Operation.Profile_torque_mode;
								PDO.Target_torque := 100; 	// Asssumed unit is in Promill
								Target_State := E_Statemachine_State.Operation_enabled;
								e_Controlword_Send := Wait_For_Send;
								e_Stop_Testing_State_Machine := Check_Start_Drive_Condition;
							END_IF	
				END_CASE
				e_Start_Type := Start_After_Reset;
				
		//__________________Check Drive Condition SM_____________________________
			Check_Start_Drive_Condition:
				// Wait for desired speed 
				IF CheckStartDelayTimer.Q THEN
					Check_Start_Delay_Timer := FALSE;  // Kann zu problemen führen, da falls der timer gleich resettet wird auch der programmzeiger nichtmehr in die If reinhüpft
					CASE e_Operation_Mode OF
						//-----------------------------------------------------------
						E_Mode_of_operation.Profile_position_mode, E_Mode_of_operation.Velocity_mode, E_Mode_of_operation.Profile_velocity_mode:
							CASE e_Start_Type OF
								Start_After_Reset:
									IF ABS(Actual_Velocity_RPM - JST_Profile_velocity_parameters.Target_velocity) < Vel_Tolerance THEN
									  // AND PDO.Statusword = E_Statusword_Bits.Target_reached THEN  //hier nochmal nachschauen
											// e_Stop_Mode muss mitgeloggt werden!!! sonst erkennt man nicht in welchem fall der motor wieder anläuft
											GLB.Logger.Message := J_Make_Message( Testing_Mode := e_Stop_Mode,
																					  Operation_Mode := e_Operation_Mode,
																				      Desired_Value := JST_Profile_velocity_parameters.Target_velocity,
																				      Real_Value := TO_INT(Actual_Velocity_RPM),
																				      Ranking := J_E_Test_Ranking.OK,
																				      Comment := 'Drive started in toleran'); 									   
											ADSLOGSTR(msgCtrlMask := ADSLOG_MSGTYPE_ERROR OR ADSLOG_MSGTYPE_LOG,
													msgFmtStr := CONCAT('Geschwindigkeit passt  ',TO_STRING(Actual_Velocity_RPM)),
													strArg := '');
											e_Stop_Testing_State_Machine := Change_Stop_Testing_State;
									
									ELSIF ABS(Actual_Velocity_RPM - JST_Profile_velocity_parameters.Target_velocity) < Vel_Tolerance THEN
										J_Make_Message(Testing_Mode := e_Stop_Mode,
														   Operation_Mode := e_Operation_Mode,
														   Desired_Value := JST_Profile_velocity_parameters.Target_velocity,
														   Real_Value := TO_INT(Actual_Velocity_RPM),
														   Ranking := J_E_Test_Ranking.Not_OK,
														   Comment := 'Drive started not in tolerance');
										ADSLOGSTR(msgCtrlMask := ADSLOG_MSGTYPE_ERROR OR ADSLOG_MSGTYPE_LOG,
												msgFmtStr := 'Nicht wieder angelaufen zefigs',
												strArg := '');
										Target_State := E_Statemachine_State.Switch_on_disabled;
										e_Controlword_Send := Wait_For_Send;
										e_Stop_Testing_State_Machine := Start_Drive;
		
									ELSIF PDO.Statusword = E_Statusword_Bits.Fault THEN // auch nochmal checken ob das so passt
										GLB.Logger.Message :=J_Make_Message(Testing_Mode := e_Stop_Mode,
																		    Operation_Mode := e_Operation_Mode,
																		    Desired_Value := JST_Profile_velocity_parameters.Target_velocity,
																		    Real_Value := TO_INT(Actual_Velocity_RPM),
																		    Ranking := J_E_Test_Ranking.Not_OK,
															   				Comment := 'Fault');
										ADSLOGSTR(msgCtrlMask := ADSLOG_MSGTYPE_ERROR OR ADSLOG_MSGTYPE_LOG,
												msgFmtStr := 'irgend ein fehler',
												strArg := '');
										Target_State := E_Statemachine_State.Switch_on_disabled;
										e_Controlword_Send := Wait_For_Send;
										e_Stop_Testing_State_Machine := Start_Drive;
									END_IF
									
								//---After Quickstop and STO stopping the drive is not supposed to run with reset
								No_Start_After_Reset:	
									IF ABS(Actual_Velocity_RPM) < Stop_Tolerance THEN
										J_Make_Message(Testing_Mode := e_Stop_Mode,
														   Operation_Mode := e_Operation_Mode,
														   Desired_Value := 0,
														   Real_Value := TO_INT(Actual_Velocity_RPM),
														   Ranking := J_E_Test_Ranking.OK,
														   Comment := 'Its not supposed to start');
										ADSLOGSTR(msgCtrlMask := ADSLOG_MSGTYPE_ERROR OR ADSLOG_MSGTYPE_LOG,
												  msgFmtStr := 'No Start after reset, passt',
												  strArg := '');
										
									ELSIF ABS(Actual_Velocity_RPM) > Stop_Tolerance THEN 
										J_Make_Message(Testing_Mode := e_Stop_Mode,
														   Operation_Mode := e_Operation_Mode,
														   Desired_Value := 0,
														   Real_Value := TO_INT(Actual_Velocity_RPM),
														   Ranking := J_E_Test_Ranking.Not_OK,
														   Comment := 'Its not supposed to start');
										ADSLOGSTR(msgCtrlMask := ADSLOG_MSGTYPE_ERROR OR ADSLOG_MSGTYPE_LOG,
											msgFmtStr := 'Start after reset passt nicht !',
											strArg := '');
									END_IF
									
									// After check for running the Drive needs to start again
									// Kann man zusammen fassen da STO1 und 2 schon gesetzt wurden unten
									IF e_Stop_Mode = J_E_Stop_Modes.Quick_Stop THEN  // Reset for quickstop
											Target_State := E_Statemachine_State.Operation_enabled;
											e_Controlword_Send := Wait_For_Send;
											Check_Start_Delay_Timer := TRUE;	
	
									ELSIF e_Stop_Mode = J_E_Stop_Modes.STO1  OR e_Stop_Mode = J_E_Stop_Modes.STO2 THEN
										Target_State := E_Statemachine_State.Operation_enabled;
										e_Controlword_Send := Wait_For_Send;
										Check_Start_Delay_Timer := TRUE;
									END_IF	
									e_Start_Type := Start_After_Reset;
								END_CASE
							
						E_Mode_of_operation.Profile_torque_mode: // muss man nochmal liebe angedeihen lassen
							// check torque
							IF PDO.Statusword = E_Statusword_Bits.Target_reached THEN
								IF Actual_Velocity_RPM > 3000 THEN
									(*fb_Message_Logging(Testing_Mode := 'Check_Start_Drive_Condition',
													   Operation_Mode := e_Operation_Mode,
													   Desired_Value := 3000,
													   Real_Value := TO_INT(Actual_Velocity_RPM),
													   Ranking := J_E_Test_Ranking.OK,
													   Comment := 'Drive started with 200 Promill Torque');*)
													   
									e_Stop_Testing_State_Machine := Stop_Testing;
												   
								ELSIF Actual_Velocity_RPM < 3000 THEN
									(*fb_Message_Logging(Testing_Mode := 'Check_Start_Drive_Condition',
													   Operation_Mode := e_Operation_Mode,
													   Desired_Value := 3000,
													   Real_Value := TO_INT(Actual_Velocity_RPM),
													   Ranking := J_E_Test_Ranking.OK,
													   Comment := 'Drive no 200 Promill Torque');*)
								END_IF
							END_IF
					END_CASE
				END_IF
		//____________ _____Change Stop testing State____________________________	
			Change_Stop_Testing_State:
					CASE e_Stop_Mode OF
						J_E_Stop_Modes.Switch_On			:	e_Stop_Mode := J_E_Stop_Modes.Shutdown;			
						J_E_Stop_Modes.Shutdown				:	e_Stop_Mode := J_E_Stop_Modes.Switch_On_Disabled;	
						J_E_Stop_Modes.Switch_On_Disabled	:	e_Stop_Mode := J_E_Stop_Modes.Vel_To_Zero;
						J_E_Stop_Modes.Vel_To_Zero			:	e_Stop_Mode := J_E_Stop_Modes.Halt;
						J_E_Stop_Modes.Halt					:	e_Stop_Mode := J_E_Stop_Modes.Quick_Stop;
						J_E_Stop_Modes.Quick_Stop			:   e_Stop_Mode := J_E_Stop_Modes.STO1;
						J_E_Stop_Modes.STO1					:	e_Stop_Mode := J_E_Stop_Modes.STO2;
						J_E_Stop_Modes.STO2					:	e_Stop_Mode := J_E_Stop_Modes.Switch_On;		
						//J_E_Stop_Modes.Fault				:	e_Stop_Mode := J_E_Stop_Modes.Switch_On;
					END_CASE
					e_Stop_Testing_State_Machine := Stop_Testing;
		//__________________Stop Testing SM______________________________________		
			Stop_Testing:

				CASE e_Operation_Mode OF
				//----------testing in Profile Position Mode---------------------
					E_Mode_of_operation.Profile_position_mode, E_Mode_of_operation.Velocity_mode, 
					E_Mode_of_operation.Profile_velocity_mode, E_Mode_of_operation.Profile_torque_mode:      // Case kann man eigenlich weglassen, da in jedem mode gleich
						//-------------------------------------------------------
						CASE e_Stop_Mode OF
						//Trigger Stopp and start timer
							J_E_Stop_Modes.Switch_On:
								//JST_Controlword := CONTROLWORD_STATE_CHANGE(JST_Current_State, E_statemachine_state.Switched_on);	
								Target_State := E_Statemachine_State.Switched_on;					
								Stop_Timer := TRUE;
								e_Stop_Type := Idle_Output_Stage;
								ADSLOGSTR(msgCtrlMask := ADSLOG_MSGTYPE_ERROR OR ADSLOG_MSGTYPE_LOG,
						  						msgFmtStr := 'Switch on',
						  						strArg := '');
								
							J_E_Stop_Modes.Shutdown:
								//JST_Controlword := CONTROLWORD_STATE_CHANGE(JST_Current_State, E_statemachine_state.Ready_to_switch_on);		
								Target_State := E_Statemachine_State.Ready_to_switch_on;				
								Stop_Timer := TRUE;
								e_Stop_Type := Idle_Output_Stage;
								ADSLOGSTR(msgCtrlMask := ADSLOG_MSGTYPE_ERROR OR ADSLOG_MSGTYPE_LOG,
						  						msgFmtStr := 'Shutdown',
						  						strArg := '');
								
							J_E_Stop_Modes.Switch_On_Disabled:
								//JST_Controlword := CONTROLWORD_STATE_CHANGE(JST_Current_State, E_statemachine_state.Switch_on_disabled);	
								Target_State := E_Statemachine_State.Switch_on_disabled;					
								Stop_Timer := TRUE;
								e_Stop_Type := Idle_Output_Stage;
								ADSLOGSTR(msgCtrlMask := ADSLOG_MSGTYPE_ERROR OR ADSLOG_MSGTYPE_LOG,
						  						msgFmtStr := 'Switch_On_Disabled',
						  						strArg := '');
								
							J_E_Stop_Modes.Vel_To_Zero: //  Torque to Zero
								PDO.Target_velocity := 0; // idk if Target or profile velocity
								PDO.vl_target_velocity := 0;
								PDO.Profile_velocity := 0;
								PDO.Target_torque := 0;
								Stop_Timer := TRUE;
								IF e_Operation_Mode = E_Mode_of_operation.Profile_position_mode OR e_Operation_Mode = E_Mode_of_operation.Profile_velocity_mode THEN
									e_Stop_Type := Vel_Zero; // was passiert hier im Torque mode?
								ELSIF e_Operation_Mode = E_Mode_of_operation.Velocity_mode THEN
									e_Stop_Type := Ramp_Down_AFAP;
								ELSIF e_Operation_Mode = E_Mode_of_operation.Profile_torque_mode THEN
									e_Stop_Type := Idle_Output_Stage;
								END_IF
								ADSLOGSTR(msgCtrlMask := ADSLOG_MSGTYPE_ERROR OR ADSLOG_MSGTYPE_LOG,
						  						msgFmtStr := 'Vel_To_Zero',
						  						strArg := '');
							J_E_Stop_Modes.Halt:
								//Trigger Stopp
								JST_Controlword := JST_Controlword OR E_Controlword_Bits.Halt;
								Send_Controlword_Direct := TRUE;
								StopTimer(PT := Stop_Time_AFAP + T#200MS );
								Stop_Timer := TRUE;
								e_Stop_Type := Ramp_Down_AFAP;	
								ADSLOGSTR(msgCtrlMask := ADSLOG_MSGTYPE_ERROR OR ADSLOG_MSGTYPE_LOG,
						  						msgFmtStr := 'Halt',
						  						strArg := '');
							J_E_Stop_Modes.Quick_Stop:
								//Trigger Stopp
								//JST_Controlword := CONTROLWORD_STATE_CHANGE(JST_Current_State, E_statemachine_state.Quick_stop_active);
								Target_State := E_Statemachine_State.Quick_stop_active;
								StopTimer(PT := T#15000MS );
								Stop_Timer := TRUE;
								e_Stop_Type := Ramp_Down_AFAP;
								ADSLOGSTR(msgCtrlMask := ADSLOG_MSGTYPE_ERROR OR ADSLOG_MSGTYPE_LOG,
						  						msgFmtStr := 'Quick_Stop',
						  						strArg := '');
								
							J_E_Stop_Modes.STO1:
								//Trigger Stopp
								OutputSTO1 := FALSE;
								Stop_Timer := TRUE;
								e_Stop_Type := Idle_Output_Stage;
								ADSLOGSTR(msgCtrlMask := ADSLOG_MSGTYPE_ERROR OR ADSLOG_MSGTYPE_LOG,
						  						msgFmtStr := 'STO1',
						  						strArg := '');
		
							J_E_Stop_Modes.STO2:
								//Trigger Stopp
								OutputSTO2 := FALSE;
								Stop_Timer := TRUE;
								e_Stop_Type := Idle_Output_Stage;
								ADSLOGSTR(msgCtrlMask := ADSLOG_MSGTYPE_ERROR OR ADSLOG_MSGTYPE_LOG,
						  						msgFmtStr := 'STO2',
						  						strArg := '');
												
							J_E_Stop_Modes.Fault: // Ideen sammeln wie man einen Fehler schmeißt
								//Trigger Stopp 																															// hier geht es morgen weiter
								//JST_Controlword := CONTROLWORD_STATE_CHANGE(JST_Current_State, E_statemachine_state.Fault);
								Target_State := E_Statemachine_State.Fault;
								StopTimer(PT := Toff);
								Stop_Timer := TRUE;
								e_Stop_Type := Idle_Output_Stage;
								ADSLOGSTR(msgCtrlMask := ADSLOG_MSGTYPE_ERROR OR ADSLOG_MSGTYPE_LOG,
						  						msgFmtStr := 'Fault',
						  						strArg := '');
						END_CASE
						
						e_Stop_Testing_State_Machine := Check_Stop_Drive_Condition;
						e_Controlword_Send := Wait_For_Send;
				END_CASE
				
				
		//________________________Check Drive Stop_______________________________		
			Check_Stop_Drive_Condition:
				
				CASE e_Stop_Type OF
					
					Idle_Output_Stage:
						// Check for Idle
						IF ABS(Actual_Velocity_RPM) < Stop_Tolerance AND StopTimer.Q = FALSE THEN
							Stop_Timer := FALSE;
							J_Make_Message(Testing_Mode := e_Stop_Mode,
											   Operation_Mode := e_Operation_Mode,
											   Desired_Value := TIME_TO_INT(Toff),
											   Real_Value := TIME_TO_INT(Elapsed_Time),
											   Ranking := J_E_Test_Ranking.OK,
											   Comment := 'PowerStage enabled, Vel=0 in < 2s');
							ADSLOGSTR(msgCtrlMask := ADSLOG_MSGTYPE_ERROR OR ADSLOG_MSGTYPE_LOG,
						  						msgFmtStr := 'PowerStage enabled, Vel=0 in < 2s',
						  						strArg := '');
							e_Stop_Testing_State_Machine := Start_Drive;
						   
						ELSIF StopTimer.Q = TRUE AND ABS(Actual_Velocity_RPM) > Stop_Tolerance  THEN
							Stop_Timer:= FALSE;
							J_Make_Message(Testing_Mode := e_Stop_Mode,
											   Operation_Mode := e_Operation_Mode,
											   Desired_Value := TIME_TO_INT(Toff),
											   Real_Value := TIME_TO_INT(Elapsed_Time),
											   Ranking := J_E_Test_Ranking.Issues,
											   Comment := 'PowerStage enabled, Vel>0 after 2s');
							ADSLOGSTR(msgCtrlMask := ADSLOG_MSGTYPE_ERROR OR ADSLOG_MSGTYPE_LOG,
						  						msgFmtStr := 'PowerStage enabled, Vel>0 in < 2s',
						  						strArg := '');
							e_Stop_Testing_State_Machine := Start_Drive;
					
						ELSIF StopTimer.Q = TRUE AND ABS(Actual_Velocity_RPM) < Stop_Tolerance  THEN
							Stop_Timer := FALSE;
							J_Make_Message(Testing_Mode := e_Stop_Mode,
											   Operation_Mode := e_Operation_Mode,
											   Desired_Value := TIME_TO_INT(Toff),
											   Real_Value := TIME_TO_INT(Elapsed_Time),
											   Ranking := J_E_Test_Ranking.Issues,
											   Comment := 'PowerStage enabled, Vel=0 after 2s');
							ADSLOGSTR(msgCtrlMask := ADSLOG_MSGTYPE_ERROR OR ADSLOG_MSGTYPE_LOG,
						  						msgFmtStr := 'PowerStage enabled, Vel=0 in 2s',
						  						strArg := '');
							e_Stop_Testing_State_Machine := Start_Drive;
						ELSE
							;
						END_IF
					//--------------------------------------------------------------	
					Ramp_Down_AFAP:
						IF StopTimer.Q = FALSE AND Actual_Velocity_RPM < Stop_Tolerance THEN
								J_Make_Message(Testing_Mode := e_Stop_Mode,
												   Operation_Mode := e_Operation_Mode,
												   Desired_Value := TIME_TO_INT(Stop_Time_AFAP),
												   Real_Value := TIME_TO_INT(Elapsed_Time),
												   Ranking := J_E_Test_Ranking.OK,
												   Comment := 'Time to Ramp Down < 500MS');
								ADSLOGSTR(msgCtrlMask := ADSLOG_MSGTYPE_ERROR OR ADSLOG_MSGTYPE_LOG,
						  						msgFmtStr := 'Time to Ramp Down < 500MS',
						  						strArg := '');
								e_Stop_Testing_State_Machine := Start_Drive;
								Stop_Timer := FALSE;

						ELSIF StopTimer.Q = TRUE AND Actual_Velocity_RPM < Stop_Tolerance THEN
								J_Make_Message(Testing_Mode := e_Stop_Mode,
												   Operation_Mode := e_Operation_Mode,
												   Desired_Value := TIME_TO_INT(Stop_Time_AFAP),
												   Real_Value := TIME_TO_INT(Elapsed_Time),
												   Ranking := J_E_Test_Ranking.Not_OK,
												   Comment := 'Time to Ramp Down > 500MS ');
								ADSLOGSTR(msgCtrlMask := ADSLOG_MSGTYPE_ERROR OR ADSLOG_MSGTYPE_LOG,
						  						msgFmtStr := 'Time to Ramp Down > 500MS',
						  						strArg := '');
								e_Stop_Testing_State_Machine := Start_Drive;
								Stop_Timer := FALSE;
								
						ELSIF StopTimer.Q = TRUE AND Actual_Velocity_RPM > Stop_Tolerance THEN
								J_Make_Message(Testing_Mode := e_Stop_Mode,
												   Operation_Mode := e_Operation_Mode,
												   Desired_Value := TIME_TO_INT(Stop_Time_AFAP),
												   Real_Value := TIME_TO_INT(Elapsed_Time),
												   Ranking := J_E_Test_Ranking.Not_OK,
												   Comment := 'No Ramp Down');
								ADSLOGSTR(msgCtrlMask := ADSLOG_MSGTYPE_ERROR OR ADSLOG_MSGTYPE_LOG,
						  						msgFmtStr := 'No Ramp Down',
						  						strArg := '');
								e_Stop_Testing_State_Machine := Start_Drive;
								Stop_Timer := FALSE;
						END_IF
					//--------------------------------------------------------------
					Vel_Zero:
						//-------------------Profile Position Mode------------------
						IF e_Operation_Mode = E_Mode_of_operation.Profile_position_mode AND StopTimer.Q = TRUE THEN
							IF ABS(Actual_Velocity_RPM - JST_Profile_velocity_parameters.Target_velocity) < Vel_Tolerance THEN
								J_Make_Message(Testing_Mode := e_Stop_Mode,
												   Operation_Mode := e_Operation_Mode,
												   Desired_Value := TO_INT(JST_Profile_velocity_parameters.Target_velocity),
												   Real_Value := TO_INT(Actual_Velocity_RPM),
												   Ranking := J_E_Test_Ranking.OK,
												   Comment := 'No velocity Zero in PPM');
								ADSLOGSTR(msgCtrlMask := ADSLOG_MSGTYPE_ERROR OR ADSLOG_MSGTYPE_LOG,
						  						msgFmtStr := 'No velocity Zero in PPM',
						  						strArg := '');
								e_Stop_Testing_State_Machine := Start_Drive;	
								Stop_Timer := FALSE;						   
							ELSIF (Actual_Velocity_RPM - JST_Profile_velocity_parameters.Target_velocity) > Vel_Tolerance THEN			//Nachdenken
								J_Make_Message(Testing_Mode := e_Stop_Mode,
												   Operation_Mode := e_Operation_Mode,
												   Desired_Value := TO_INT(JST_Profile_velocity_parameters.Target_velocity),
												   Real_Value := TO_INT(Actual_Velocity_RPM),
												   Ranking := J_E_Test_Ranking.OK,
												   Comment := 'No velocity Zero in PPM');
								ADSLOGSTR(msgCtrlMask := ADSLOG_MSGTYPE_ERROR OR ADSLOG_MSGTYPE_LOG,
						  						msgFmtStr := 'No velocity Zero in PPM',
						  						strArg := '');
								e_Stop_Testing_State_Machine := Start_Drive;
								Stop_Timer := FALSE;
							ELSE
								J_Make_Message(Testing_Mode := e_Stop_Mode,
												   Operation_Mode := e_Operation_Mode,
												   Desired_Value := TO_INT(JST_Profile_velocity_parameters.Target_velocity),
												   Real_Value := TO_INT(Actual_Velocity_RPM),
												   Ranking := J_E_Test_Ranking.Not_OK,
												   Comment := 'Vel not 0 and not desired value');
								ADSLOGSTR(msgCtrlMask := ADSLOG_MSGTYPE_ERROR OR ADSLOG_MSGTYPE_LOG,
						  						msgFmtStr := 'Vel not 0 and not desired value',
						  						strArg := '');
								e_Stop_Testing_State_Machine := Start_Drive;
								Stop_Timer := FALSE;
							END_IF
							
						//----------------------Profile Velocity Mode-----------------------	
						//  Test if Ramp at 50% down is ok
						ELSIF e_Operation_Mode = E_Mode_of_operation.Profile_velocity_mode AND StopTimer.Q = FALSE THEN
							IF ABS(Actual_Velocity_RPM - JST_Profile_velocity_parameters.Target_velocity/2) < Vel_Tolerance THEN
								StopTimer(ET => Elapsed_Time);
								IF TO_DWORD(Time_Tolerance) > ABS(TO_DWORD(Elapsed_Time)-TO_DWORD(JST_Profile_velocity_parameters.Target_velocity)/JST_Profile_velocity_parameters.Profile_deceleration)/2 THEN
									J_Make_Message(Testing_Mode := e_Stop_Mode,
													   Operation_Mode := e_Operation_Mode,
													   Desired_Value := JST_Profile_velocity_parameters.Target_velocity/2,
													   Real_Value := TO_INT(Actual_Velocity_RPM),
													   Ranking := J_E_Test_Ranking.OK,
													   Comment := '50% Ramp Down OK');
								ELSE 
									J_Make_Message(Testing_Mode := e_Stop_Mode,
													   Operation_Mode := e_Operation_Mode,
													   Desired_Value := JST_Profile_velocity_parameters.Target_velocity,
													   Real_Value := TO_INT(Actual_Velocity_RPM),
													   Ranking := J_E_Test_Ranking.Not_OK,
													   Comment := '50% Ramp Down not OK');
									e_Stop_Testing_State_Machine := Start_Drive;
								END_IF
							// check if ramp at 100% (vel = 0) is ok
							ELSIF ABS(Actual_Velocity_RPM) < Vel_Tolerance AND StopTimer.Q = FALSE THEN
								Stop_Timer := FALSE;
								IF TO_DWORD(Time_Tolerance) > ABS(TO_DWORD(Elapsed_Time)-TO_DWORD(JST_Profile_velocity_parameters.Target_velocity)/JST_Profile_velocity_parameters.Profile_deceleration)/2 THEN
									J_Make_Message(Testing_Mode := e_Stop_Mode,
													   Operation_Mode := e_Operation_Mode,
													   Desired_Value := JST_Profile_velocity_parameters.Target_velocity/2,
													   Real_Value := TO_INT(Actual_Velocity_RPM),
													   Ranking := J_E_Test_Ranking.OK,
													   Comment := '100% Ramp Down OK');
								ELSE 
									J_Make_Message(Testing_Mode := e_Stop_Mode,
													   Operation_Mode := e_Operation_Mode,
													   Desired_Value := JST_Profile_velocity_parameters.Target_velocity,
													   Real_Value := TO_INT(Actual_Velocity_RPM),
													   Ranking := J_E_Test_Ranking.Not_OK,
													   Comment := '100% Ramp Down NOT OK');
									e_Stop_Testing_State_Machine := Start_Drive;
								END_IF
							ELSE 
								//Timeout ramp longer than 2sec
								J_Make_Message(Testing_Mode := e_Stop_Mode,
														   Operation_Mode := E_Mode_of_operation.Profile_velocity_mode,
														   Desired_Value := JST_Profile_velocity_parameters.Target_velocity,
														   Real_Value := TO_INT(Actual_Velocity_RPM),
														   Ranking := J_E_Test_Ranking.Not_OK,
														   Comment := 'Time failure while ramp down');
								e_Stop_Testing_State_Machine := Start_Drive;
							END_IF
						END_IF		
				END_CASE
				
				IF e_Stop_Testing_State_Machine = Start_Drive THEN
						Start_Delay_Timer := TRUE;
				END_IF
				
		// Statechange nach Check start drive condition		
		//_____________________Start Drive Again___________________________________________	
			Start_Drive: 
				IF StartDelayTimer.Q THEN
					Start_Delay_Timer := FALSE;
					CASE e_Stop_Mode OF
						J_E_Stop_Modes.Switch_On:
							Target_State := E_Statemachine_State.Operation_enabled;	
							e_Controlword_Send := Wait_For_Send;
							//e_Stop_Mode := J_E_Stop_Modes.Shutdown;
							e_Start_Type := Start_After_Reset;					
						J_E_Stop_Modes.Shutdown:
							Target_State := E_Statemachine_State.Operation_enabled;
							e_Controlword_Send := Wait_For_Send;
							//e_Stop_Mode := J_E_Stop_Modes.Switch_On_Disabled;	
							e_Start_Type := Start_After_Reset;					
						J_E_Stop_Modes.Switch_On_Disabled:
							Target_State := E_Statemachine_State.Operation_enabled;
							e_Controlword_Send := Wait_For_Send;
							//e_Stop_Mode := J_E_Stop_Modes.Vel_To_Zero;
							e_Start_Type := Start_After_Reset;
						J_E_Stop_Modes.Vel_To_Zero:
							PDO.Target_velocity := JST_Profile_velocity_parameters.Target_velocity; // No vel to zero in PPM
							PDO.vl_target_velocity := TO_INT(JST_Profile_velocity_parameters.Target_velocity);
							//e_Stop_Mode := J_E_Stop_Modes.Halt;
							e_Start_Type := Start_After_Reset;
						J_E_Stop_Modes.Halt:
							JST_Controlword := JST_Controlword AND NOT E_Controlword_Bits.Halt;    // muss man noch schauen wie man das in die SM integriert
							Send_Controlword_Direct := TRUE;
							e_Controlword_Send := Wait_For_Send;
							//e_Stop_Mode := J_E_Stop_Modes.Quick_Stop;
							e_Start_Type := Start_After_Reset;
						J_E_Stop_Modes.Quick_Stop:
							JST_Controlword := 16#000F;
							Send_Controlword_Direct := TRUE;
							e_Controlword_Send := Wait_For_Send;
							//StopTimer(PT := T#1000MS);		//Quickstopramp to slow
							//StaStop_Timer TRUE;
							//e_Stop_Mode := J_E_Stop_Modes.STO1;
							e_Start_Type := No_Start_after_Reset;
						J_E_Stop_Modes.STO1:
							OutputSTO1 := TRUE;
							//StopTimer(IN := StaStop_Timer := T#1000MS);  // Timer fuuuu
							e_Start_Type := No_Start_after_Reset;
							//e_Stop_Mode := J_E_Stop_Modes.STO2;
						J_E_Stop_Modes.STO2:
							OutputSTO2 := TRUE;
							//StopTimer(IN := StaStop_Timer := T#1000MS);
							//e_Stop_Mode := Fault;
							e_Start_Type := No_Start_after_Reset;
							//e_Stop_Mode := J_E_Stop_Modes.Switch_On;   // Start Again
							
						J_E_Stop_Modes.Fault:
							//Start again
							//e_Start_Type := No_Start_after_Reset;
							//e_Stop_Mode := J_E_Stop_Modes.Switch_On;
					
					END_CASE
					e_Stop_Testing_State_Machine := Check_Start_Drive_Condition;
					Check_Start_Delay_Timer := TRUE;
				END_IF

		//_________________________Error Handling_______________________________
			Error_Handling:
				;
		END_CASE
		
		
		
	Wait_For_Send:
		IF NOT Send_Controlword_Direct THEN
			IF JST_Current_State = Target_State THEN
				e_Controlword_Send := Continue_SM;
			ELSE
				JST_Controlword := CONTROLWORD_STATE_CHANGE(JST_Current_State, Target_State);
				e_Controlword_Send := Wait_For_Send;
			END_IF
		ELSIF Send_Controlword_Direct THEN
			JST_Controlword := JST_Controlword;
			Send_Controlword_Direct := FALSE;
			e_Controlword_Send := Continue_SM;
		END_IF
END_CASE

END_FUNCTION_BLOCK

// ---- POUs/FUN/J_Make_Message.TcPOU
FUNCTION J_Make_Message : STRING
VAR_INPUT
	Operation_Mode : E_Mode_of_operation;
	Testing_Mode   : J_E_Stop_Modes;
	Desired_Value  : DINT;
	Real_Value     : DINT;
	Ranking 	   : J_E_Test_Ranking;
	Comment		   : STRING(256);
END_VAR
VAR
	Message : STRING;
END_VAR

Message := CONCAT(Message, TO_STRING(Operation_Mode));
Message := CONCAT(Message,',');
//Message := CONCAT(Message,'$T');
Message := CONCAT(Message, TO_STRING(Testing_Mode));
Message := CONCAT(Message,',');
//Message := CONCAT(Message,'$T');
Message := CONCAT(Message, DINT_TO_STRING(Desired_Value));
Message := CONCAT(Message,',');
//Message := CONCAT(Message,'$T');
Message := CONCAT(Message, DINT_TO_STRING(Real_Value));
Message := CONCAT(Message,',');
//Message := CONCAT(Message,'$T');
Message := CONCAT(Message, TO_STRING(Ranking));
Message := CONCAT(Message,',');
//Message := CONCAT(Message,'$T');
Message := CONCAT(Message, Comment);
Message := CONCAT(Message,'$n');

GLB.Logger.SaveFlag := TRUE;

J_Make_Message := Message;

END_FUNCTION

// ---- POUs/FB/FB_Logger.TcPOU
FUNCTION_BLOCK FB_Logger
VAR_INPUT
	NetId			: STRING		:= '10.200.20.88.1.1';	
	FileName		: STRING 		:= 'C:\LogFile.log';
	Timeout			: TIME			:= T#100MS;			// Timeout

	Message			: STRING(256)	:= '';				// Write this message with index, timestamp and a new line suffix
	OpenFlag		: BOOL			:= FALSE;			// Open the file
	CloseFlag		: BOOL			:= FALSE;			// Close the file
	SaveFlag		: BOOL			:= FALSE;			// Save the file
END_VAR
VAR_OUTPUT		
	State			: e_LoggerState	:= e_LoggerState.Closed;
	IsOpen			: BOOL			:= FALSE;	
END_VAR
VAR
	Open			: FB_FileOpen;
	Write			: FB_FilePuts;
	Close   		: FB_FileClose;

	Index			: DWORD			:= 1;
	MessageBuffer	: STRING 		:= '';
	
    GetSystemTime 	: GETSYSTEMTIME;
    StartFileTime   : T_FILETIME;
	FileTime   		: T_FILETIME;	
    SystemTime		: TIMESTRUCT;
    Filedate 		: STRING(15)	:= '';
	Startdate		: STRING(20);
    Timestamp 		: STRING(30);
END_VAR

// Add the new message to write
IF (Message <> '') THEN
	IF Filedate = '' THEN
		Timestamp := '0';		
	ELSE
		// Timestamp with format: YHH:MM:SS.mmm		
		GetSystemTime(timeLoDW => FileTime.dwLowDateTime, timeHiDW => FileTime.dwHighDateTime);
		Timestamp := LINT_TO_STRING((SHL(DWORD_TO_LINT(FileTime.dwHighDateTime), 32) + DWORD_TO_LINT(FileTime.dwLowDateTime) - SHL(DWORD_TO_LINT(StartFileTime.dwHighDateTime), 32) - DWORD_TO_LINT(StartFileTime.dwLowDateTime))/10000);	
	END_IF	
	MessageBuffer := CONCAT(CONCAT(CONCAT(CONCAT(CONCAT(CONCAT(MessageBuffer, DWORD_TO_STRING(Index)), ';'), Timestamp), ';'), Message), '$0A');	
	Index := Index + 1;
	Message := '';
END_IF



CASE State OF
	// ***** Open the logger file *****
	e_LoggerState.Open:
		IF IsOpen THEN
			// The logger file is already opened			
			State := e_LoggerState.Opened;
		ELSIF OpenFlag OR SaveFlag THEN
			// Start opening
			IF OpenFlag THEN
				// Timestamp with format: YYYYMMDD_HHMMSS			
				GetSystemTime(timeLoDW => StartFileTime.dwLowDateTime, timeHiDW => StartFileTime.dwHighDateTime);
				SystemTime := FILETIME_TO_SYSTEMTIME(StartFileTime);
				Filedate := CONCAT(	CONCAT(	CONCAT(	CONCAT(	CONCAT(	CONCAT(	WORD_TO_STRING(SystemTime.wYear),
																			RIGHT(CONCAT('0',WORD_TO_STRING(SystemTime.wMonth)),2)),
																	RIGHT(CONCAT('0',WORD_TO_STRING(SystemTime.wDay)),2)),
															'_'),
													RIGHT(CONCAT('0',WORD_TO_STRING(SystemTime.wHour)),2)),
											RIGHT(CONCAT('0',WORD_TO_STRING(SystemTime.wMinute)),2)),
									RIGHT(CONCAT('0',WORD_TO_STRING(SystemTime.wSecond)),2));									

				// Write header	
				Startdate := CONCAT(CONCAT(	CONCAT(	CONCAT(	CONCAT(	CONCAT(	CONCAT(	RIGHT(CONCAT('0',WORD_TO_STRING(SystemTime.wDay)),2),
																					'.'),
																			CONCAT(	RIGHT(CONCAT('0',WORD_TO_STRING(SystemTime.wMonth)),2),
																					'.')),
																	WORD_TO_STRING(SystemTime.wYear)),
															' '),
													CONCAT(RIGHT(CONCAT('0',WORD_TO_STRING(SystemTime.wHour)),2),':')),
											CONCAT(RIGHT(CONCAT('0',WORD_TO_STRING(SystemTime.wMinute)),2),':')),
									RIGHT(CONCAT('0',WORD_TO_STRING(SystemTime.wSecond)),2));
				
				MessageBuffer := CONCAT(CONCAT(	CONCAT(	 'Startdate;', Startdate ), 
												'$0A$0ANo.;Timestamp [ms];Info$0A'),
										MessageBuffer);										
			END_IF
			
			Open(sNetId := NetID, 
				 sPathName := INSERT(FileName, CONCAT('_', Filedate), FIND(FileName,'.')-1), 
				 nMode := FOPEN_MODEAPPEND OR FOPEN_MODETEXT, bExecute:=TRUE, tTimeout:=Timeout);
			State := e_LoggerState.Opening;
		END_IF
		
		
	// ***** The logger file is currently opening. *****
	e_LoggerState.Opening:
		IF IsOpen THEN
			// The logger file is already opened
			State := e_LoggerState.Opened;			
		ELSE
			Open(bExecute:=FALSE);
			IF NOT Open.bBusy THEN
				IF Open.hFile <> 0 THEN
					// Opening is finished
					Write(sNetId:=Open.sNetId, hFile:=Open.hFile, bExecute:=FALSE);
					Close(sNetId:=Open.sNetId, hFile:=Open.hFile, bExecute:=FALSE);					
					IsOpen := TRUE;	
					IF OpenFlag THEN 
						OpenFlag := FALSE;
					ELSE
						SaveFlag := FALSE; 
					END_IF			
					State := e_LoggerState.Opened;	
				ELSE
					// Open function is not busy but no file is opened
					State := e_LoggerState.Closed;					
				END_IF		
			ELSIF Open.bError THEN
				// Error
				State := e_LoggerState.Opening_Error;
			END_IF		
		END_IF
		
		
	// ***** A error at opening logger file has occured *****		
	e_LoggerState.Opening_Error:	
		ADSLOGSTR(msgCtrlMask := ADSLOG_MSGTYPE_ERROR OR ADSLOG_MSGTYPE_MSGBOX,
				  msgFmtStr := 'Error during opening the logger file: %s',
				  strArg := TO_STRING(Open.nErrId));
		State := e_LoggerState.Closed;
	
				  
	// ***** The logger file is opened and write data as required. *****
	e_LoggerState.Opened:
		IF Close.bBusy THEN
			// Closing is already startet (external triggered)
			State := e_LoggerState.Closing;					
		ELSIF Write.bBusy THEN
			// Writing is runing (external triggered)
			State := e_LoggerState.Writing;				
		ELSE					
			// String to write is exists -> Start writing
			IF MessageBuffer <> '' THEN	
				Close(bExecute:=FALSE);	
				Write(sLine:=MessageBuffer, bExecute:=TRUE, tTimeout:=Timeout);		
				MessageBuffer := '';		
				State := e_LoggerState.Writing;				
			ELSE		
				IF CloseFlag OR SaveFlag THEN
					// Close command
					State := e_LoggerState.Close;	
				END_IF
			END_IF;
		END_IF
	
		
	// ***** Writing to the logger file *****	
	e_LoggerState.Writing:
		Write(bExecute:=FALSE);		
		IF NOT Write.bBusy THEN
			// Writing is completed
			Write(bExecute:=FALSE);	
			State := e_LoggerState.Opened;
		ELSIF Write.bError THEN
			// An error has occured
			State := e_LoggerState.Writing_Error;
		END_IF
		
				
	// ***** A error at writing to logger file has occured *****		
	e_LoggerState.Writing_Error:	
		ADSLOGSTR(msgCtrlMask := ADSLOG_MSGTYPE_ERROR OR ADSLOG_MSGTYPE_MSGBOX,
				  msgFmtStr := 'Error during writing to the logger file: %s',
				  strArg := TO_STRING(Write.nErrId));
		State := e_LoggerState.Opened;	
			  
		
	// ***** Close the logger file *****	
	e_LoggerState.Close:
		IF IsOpen THEN	
			// Start closing
			Close(bExecute:=TRUE, tTimeout:=Timeout);
			State := e_LoggerState.Closing;
		ELSE
			// The logger file is already closed			
			State := e_LoggerState.Closed;
		END_IF
				
		
	// ***** The logger file is currently closing *****
	e_LoggerState.Closing:	
		IF IsOpen THEN
			Close(bExecute:=FALSE);
			IF NOT Close.bBusy THEN
				// Closing is finished
				IF CloseFlag THEN			
					// If the command is save and close then the close command is enough.
					IF SaveFlag THEN SaveFlag := FALSE; END_IF
					Index := 1;
					Filedate := '';
					CloseFlag := FALSE;
				END_IF;
				State := e_LoggerState.Closed;
			ELSIF Close.bError THEN
				// Error
				State := e_LoggerState.Closing_Error;
			END_IF
		ELSE
			// The logger file is already closed
			State := e_LoggerState.Closed;
		END_IF		
	
		
	// ***** A error at closing logger file has occured *****		
	e_LoggerState.Closing_Error:	
		ADSLOGSTR(msgCtrlMask := ADSLOG_MSGTYPE_ERROR OR ADSLOG_MSGTYPE_MSGBOX,
				  msgFmtStr := 'Error during closing the logger file: %s',
				  strArg := TO_STRING(Close.nErrId));
		State := e_LoggerState.Opened;			
				  
		
	// ***** The logger file is closed *****
	e_LoggerState.Closed:	
		IsOpen := FALSE;	
		
		// Check, if the open function is triggered
		IF OpenFlag OR SaveFlag OR Open.bBusy THEN
			State := e_LoggerState.Open;	
		ELSE
			CloseFlag := FALSE;
		END_IF
	
END_CASE

END_FUNCTION_BLOCK

// ---- POUs/FB/Basic/FB_SDO_WRITE_REAL.TcPOU
FUNCTION_BLOCK FB_SDO_WRITE_REAL
VAR_INPUT
	ADSNetID		: STRING(23); 	(* The AMSNetID addresses the EL6751. Can be empty if only one local single channel card is present*)
	PortNr			: WORD; 		(* The Port No. addresses the CANopen Node (see System Manager) *)
	CO_Index		: DWORD; 		(* This is the Index of the CANopen Object Dictionary Entry*)
	CO_SubIndex		: DWORD; 		(* This is the Sub-Index of the CANopen Object Dictionary Entry*)
	StartWriting	: BOOL; 		(* only reset to FALSE after WriteDataFinished=TRUE*)
	WriteData		: REAL; 		(* This real variable contains the data to be written to the CANopen Object Dictionary*)
END_VAR
VAR_OUTPUT
	WriteDataFinished	: BOOL;
	Error			: DWORD;
END_VAR
VAR
	state			: BYTE := 0;
	ADSWRITE		: ADSWRITE;
END_VAR

CASE
state OF
0:
	IF StartWriting THEN
		WriteDataFinished := FALSE;
		Error := 0;
		ADSWrite(
			NETID	:= ADSNetID,
			PORT	:= PortNr,
			IDXGRP	:= CO_Index,
			IDXOFFS	:= CO_SubIndex,
			LEN		:= 4,
			SRCADDR	:= ADR(WriteData),
			WRITE	:= TRUE,
			TMOUT 	:= T#100MS
		);
		IF ADSWrite.err THEN
			state := 2;
			WriteDataFinished := TRUE;
			Error := ADSWrite.ErrId;
		ELSE
			state := 1;
		END_IF
	ELSE
		ADSWrite(
			NETID	:= '',
			PORT	:= PortNr,
			IDXGRP	:= CO_Index,
			IDXOFFS	:= CO_SubIndex,
			LEN		:= 4,
			SRCADDR	:= ADR(WriteData),
			WRITE	:= FALSE,
			TMOUT 	:= T#100MS
		);
	END_IF
	
1:
	ADSWrite(WRITE:= FALSE);
	IF ADSWrite.err THEN
		state := 2;
		WriteDataFinished := TRUE;
		Error := ADSWrite.ErrId;
	ELSE
		IF NOT ADSWrite.busy THEN
			state := 2;
			WriteDataFinished := TRUE;
		END_IF
	END_IF
	
2:
	ADSWrite(WRITE:= FALSE);
	state := 0;
END_CASE

END_FUNCTION_BLOCK

// ---- POUs/FUN/Get_Vel_RPM.TcPOU
FUNCTION Get_Vel_RPM : DINT
VAR_INPUT
	Increment_Per_Sec : DINT := 0;
END_VAR

Get_Vel_RPM := (Increment_Per_Sec/4096) * 60;

END_FUNCTION

// ---- POUs/WRITE_Manufacturer_label.TcPOU
FUNCTION_BLOCK WRITE_Manufacturer_label
VAR_INPUT
	Label_In	: ST_Manufacturer_label;
	NodeID		: BYTE; (* This Port No. addresses the CANopen Node (see System Manager) *)	
	Start		: BOOL;
END_VAR
VAR_OUTPUT
	Finished	: BOOL := FALSE;
END_VAR
VAR
	Index		: INT;
	Label		: ST_Manufacturer_label;
	SDO_WRITE 	: FB_SDO_WRITE;
	WriteData		: ARRAY [0..255] OF BYTE;	
	CAN_Objects: INT;
	
	fbTonDelay		: TON;
END_VAR

// Restart after complete run
IF (Index = 255) AND Start THEN
	Index := 0;
END_IF


IF NOT (Index = 255) THEN 
	SDO_WRITE(StartWriting:=FALSE);
	FB_SDO_WRITE_REAL(StartWriting:=FALSE);
END_IF


CASE Index OF	
	0: 
		IF Start THEN	
			Label := Label_In;	
			Finished := FALSE;
			WriteData[0] := DWORD_TO_BYTE(Label.Min_v);
			WriteData[1] := DWORD_TO_BYTE(SHR(Label.Min_v,8));
			WriteData[2] := DWORD_TO_BYTE(SHR(Label.Min_v,16));
			WriteData[3] := DWORD_TO_BYTE(SHR(Label.Min_v,24));		
			SDO_WRITE(	
				AdsNetID		:= GLB.ADSNetID_CAN,
				PortNr			:= 16#1000 + GLB.NodeID,
				CO_Index		:= 16#41C0,
				CO_SubIndex		:= 16#03,
				DataLength		:= 4,
				WriteData		:= WriteData,
				StartWriting	:= TRUE	
			);	
			Index := Index + 1;
		END_IF
	
	
	1: 
		IF SDO_WRITE.WriteDataFinished THEN
			WriteData[0] := DWORD_TO_BYTE(Label.Max_v);
			WriteData[1] := DWORD_TO_BYTE(SHR(Label.Max_v,8));
			WriteData[2] := DWORD_TO_BYTE(SHR(Label.Max_v,16));
			WriteData[3] := DWORD_TO_BYTE(SHR(Label.Max_v,24));		
			SDO_WRITE(	
				AdsNetID		:= GLB.ADSNetID_CAN,
				PortNr			:= 16#1000 + GLB.NodeID,
				CO_Index		:= 16#41C0,
				CO_SubIndex		:= 16#04,
				DataLength		:= 4,
				WriteData		:= WriteData,
				StartWriting	:= TRUE	
			);	
			Index := Index + 1;
		ELSE
			SDO_WRITE();
		END_IF
	
	
	2: 
		IF SDO_WRITE.WriteDataFinished THEN
			WriteData[0] := DWORD_TO_BYTE(Label.Motor_rated_current);
			WriteData[1] := DWORD_TO_BYTE(SHR(Label.Motor_rated_current,8));
			WriteData[2] := DWORD_TO_BYTE(SHR(Label.Motor_rated_current,16));
			WriteData[3] := DWORD_TO_BYTE(SHR(Label.Motor_rated_current,24));		
			SDO_WRITE(	
				AdsNetID		:= GLB.ADSNetID_CAN,
				PortNr			:= 16#1000 + GLB.NodeID,
				CO_Index		:= 16#41C0,
				CO_SubIndex		:= 16#05,
				DataLength		:= 4,
				WriteData		:= WriteData,
				StartWriting	:= TRUE	
			);	
			Index := Index + 1;
		ELSE
			SDO_WRITE();
		END_IF
	
	
	3: 
		IF SDO_WRITE.WriteDataFinished THEN
			WriteData[0] := DWORD_TO_BYTE(Label.Drive_rated_current);
			WriteData[1] := DWORD_TO_BYTE(SHR(Label.Drive_rated_current,8));
			WriteData[2] := DWORD_TO_BYTE(SHR(Label.Drive_rated_current,16));
			WriteData[3] := DWORD_TO_BYTE(SHR(Label.Drive_rated_current,24));		
			SDO_WRITE(	
				AdsNetID		:= GLB.ADSNetID_CAN,
				PortNr			:= 16#1000 + GLB.NodeID,
				CO_Index		:= 16#41C0,
				CO_SubIndex		:= 16#06,
				DataLength		:= 4,
				WriteData		:= WriteData,
				StartWriting	:= TRUE	
			);	
			Index := Index + 1;
		ELSE
			SDO_WRITE();
		END_IF
	
	
	4: 
		IF SDO_WRITE.WriteDataFinished THEN
			WriteData[0] := DWORD_TO_BYTE(Label.Max_current);
			WriteData[1] := DWORD_TO_BYTE(SHR(Label.Max_current,8));
			WriteData[2] := 0;
			WriteData[3] := 0;		
			SDO_WRITE(	
				AdsNetID		:= GLB.ADSNetID_CAN,
				PortNr			:= 16#1000 + GLB.NodeID,
				CO_Index		:= 16#41C0,
				CO_SubIndex		:= 16#07,
				DataLength		:= 2,
				WriteData		:= WriteData,
				StartWriting	:= TRUE	
			);	
			Index := Index + 1;
		ELSE
			SDO_WRITE();
		END_IF	
		
		
	5: 
		IF SDO_WRITE.WriteDataFinished THEN
			WriteData[0] := DWORD_TO_BYTE(Label.Motor_rated_torque);
			WriteData[1] := DWORD_TO_BYTE(SHR(Label.Motor_rated_torque,8));
			WriteData[2] := DWORD_TO_BYTE(SHR(Label.Motor_rated_torque,16));
			WriteData[3] := DWORD_TO_BYTE(SHR(Label.Motor_rated_torque,24));		
			SDO_WRITE(	
				AdsNetID		:= GLB.ADSNetID_CAN,
				PortNr			:= 16#1000 + GLB.NodeID,
				CO_Index		:= 16#41C0,
				CO_SubIndex		:= 16#08,
				DataLength		:= 4,
				WriteData		:= WriteData,
				StartWriting	:= TRUE	
			);	
			Index := Index + 1;
		ELSE
			SDO_WRITE();
		END_IF
	
	
	6: 
		IF SDO_WRITE.WriteDataFinished THEN
			WriteData[0] := DWORD_TO_BYTE(Label.Max_torque);
			WriteData[1] := DWORD_TO_BYTE(SHR(Label.Max_torque,8));
			WriteData[2] := 0;
			WriteData[3] := 0;		
			SDO_WRITE(	
				AdsNetID		:= GLB.ADSNetID_CAN,
				PortNr			:= 16#1000 + GLB.NodeID,
				CO_Index		:= 16#41C0,
				CO_SubIndex		:= 16#09,
				DataLength		:= 2,
				WriteData		:= WriteData,
				StartWriting	:= TRUE	
			);	
			Index := Index + 1;
		ELSE
			SDO_WRITE();
		END_IF
			
		
	7: 
		IF SDO_WRITE.WriteDataFinished THEN
			WriteData[0] := DWORD_TO_BYTE(Label.Motor_rated_speed);
			WriteData[1] := DWORD_TO_BYTE(SHR(Label.Motor_rated_speed,8));
			WriteData[2] := DWORD_TO_BYTE(SHR(Label.Motor_rated_speed,16));
			WriteData[3] := DWORD_TO_BYTE(SHR(Label.Motor_rated_speed,24));		
			SDO_WRITE(	
				AdsNetID		:= GLB.ADSNetID_CAN,
				PortNr			:= 16#1000 + GLB.NodeID,
				CO_Index		:= 16#41C0,
				CO_SubIndex		:= 16#0A,
				DataLength		:= 4,
				WriteData		:= WriteData,
				StartWriting	:= TRUE	
			);	
			Index := Index + 1;
		ELSE
			SDO_WRITE();
		END_IF
	
		
	8: 
		IF SDO_WRITE.WriteDataFinished THEN
			WriteData[0] := DWORD_TO_BYTE(Label.Number_of_pole_pairs);
			WriteData[1] := DWORD_TO_BYTE(SHR(Label.Number_of_pole_pairs,8));
			WriteData[2] := 0;
			WriteData[3] := 0;		
			SDO_WRITE(	
				AdsNetID		:= GLB.ADSNetID_CAN,
				PortNr			:= 16#1000 + GLB.NodeID,
				CO_Index		:= 16#41C0,
				CO_SubIndex		:= 16#0B,
				DataLength		:= 2,
				WriteData		:= WriteData,
				StartWriting	:= TRUE	
			);	
			Index := Index + 1;
		ELSE
			SDO_WRITE();
		END_IF
			
		
	9: 
		IF SDO_WRITE.WriteDataFinished THEN
			FB_SDO_WRITE_REAL(	
				AdsNetID		:= GLB.ADSNetID_CAN,
				PortNr			:= 16#1000 + GLB.NodeID,
				CO_Index		:= 16#41C0,
				CO_SubIndex		:= 16#0C,
				WriteData		:= Label.Motor_torque_constant,
				StartWriting	:= TRUE	
			);	
			Index := Index + 1;
		ELSE
			SDO_WRITE();
		END_IF
			
		
	10: 
		IF FB_SDO_WRITE_REAL.WriteDataFinished THEN
			FB_SDO_WRITE_REAL(	
				AdsNetID		:= GLB.ADSNetID_CAN,
				PortNr			:= 16#1000 + GLB.NodeID,
				CO_Index		:= 16#41C0,
				CO_SubIndex		:= 16#0D,
				WriteData		:= Label.Flux_producing_P_gain,
				StartWriting	:= TRUE	
			);	
			Index := Index + 1;
		ELSE
			FB_SDO_WRITE_REAL();
		END_IF
			
		
	11: 
		IF FB_SDO_WRITE_REAL.WriteDataFinished THEN
			FB_SDO_WRITE_REAL(	
				AdsNetID		:= GLB.ADSNetID_CAN,
				PortNr			:= 16#1000 + GLB.NodeID,
				CO_Index		:= 16#41C0,
				CO_SubIndex		:= 16#0E,
				WriteData		:= Label.Flux_producing_I_gain,
				StartWriting	:= TRUE	
			);	
			Index := Index + 1;
		ELSE
			FB_SDO_WRITE_REAL();
		END_IF
			
		
	12: 
		IF FB_SDO_WRITE_REAL.WriteDataFinished THEN	
			FB_SDO_WRITE_REAL(	
				AdsNetID		:= GLB.ADSNetID_CAN,
				PortNr			:= 16#1000 + GLB.NodeID,
				CO_Index		:= 16#41C0,
				CO_SubIndex		:= 16#0F,
				WriteData		:= Label.Torque_producing_P_gain,
				StartWriting	:= TRUE	
			);	
			Index := Index + 1;
		ELSE
			FB_SDO_WRITE_REAL();
		END_IF
			
		
	13: 
		IF FB_SDO_WRITE_REAL.WriteDataFinished THEN
			FB_SDO_WRITE_REAL(	
				AdsNetID		:= GLB.ADSNetID_CAN,
				PortNr			:= 16#1000 + GLB.NodeID,
				CO_Index		:= 16#41C0,
				CO_SubIndex		:= 16#10,
				WriteData		:= Label.Torque_producing_I_gain,
				StartWriting	:= TRUE	
			);	
			Index := Index + 1;
		ELSE
			FB_SDO_WRITE_REAL();
		END_IF
			
		
	14: 
		IF FB_SDO_WRITE_REAL.WriteDataFinished THEN
			WriteData[0] := DWORD_TO_BYTE(Label.Magnetic_encoder_offset);
			WriteData[1] := DWORD_TO_BYTE(SHR(Label.Magnetic_encoder_offset,8));
			WriteData[2] := 0;
			WriteData[3] := 0;		
			SDO_WRITE(	
				AdsNetID		:= GLB.ADSNetID_CAN,
				PortNr			:= 16#1000 + GLB.NodeID,
				CO_Index		:= 16#41C0,
				CO_SubIndex		:= 16#11,
				DataLength		:= 2,
				WriteData		:= WriteData,
				StartWriting	:= TRUE	
			);	
			Index := Index + 1;
		ELSE
			FB_SDO_WRITE_REAL();
		END_IF
			
		
	15: 
		IF SDO_WRITE.WriteDataFinished THEN
			WriteData[0] := DWORD_TO_BYTE(Label.Motor_with_brake);
			WriteData[1] := DWORD_TO_BYTE(SHR(Label.Motor_with_brake,8));
			WriteData[2] := 0;
			WriteData[3] := 0;		
			SDO_WRITE(	
				AdsNetID		:= GLB.ADSNetID_CAN,
				PortNr			:= 16#1000 + GLB.NodeID,
				CO_Index		:= 16#41C0,
				CO_SubIndex		:= 16#12,
				DataLength		:= 2,
				WriteData		:= WriteData,
				StartWriting	:= TRUE	
			);	
			Index := Index + 1;
		ELSE
			SDO_WRITE();
		END_IF
			
		
	16: 
		IF SDO_WRITE.WriteDataFinished THEN
			WriteData[0] := DWORD_TO_BYTE(Label.Encoder_mode_adjust);
			WriteData[1] := DWORD_TO_BYTE(SHR(Label.Encoder_mode_adjust,8));
			WriteData[2] := 0;
			WriteData[3] := 0;		
			SDO_WRITE(	
				AdsNetID		:= GLB.ADSNetID_CAN,
				PortNr			:= 16#1000 + GLB.NodeID,
				CO_Index		:= 16#41C0,
				CO_SubIndex		:= 16#13,
				DataLength		:= 2,
				WriteData		:= WriteData,
				StartWriting	:= TRUE	
			);	
			Index := Index + 1;
		ELSE
			SDO_WRITE();
		END_IF
			
		
	17: 
		IF SDO_WRITE.WriteDataFinished THEN
			WriteData[0] := DWORD_TO_BYTE(Label.Motor_max_speed);
			WriteData[1] := DWORD_TO_BYTE(SHR(Label.Motor_max_speed,8));
			WriteData[2] := 0;
			WriteData[3] := 0;		
			SDO_WRITE(	
				AdsNetID		:= GLB.ADSNetID_CAN,
				PortNr			:= 16#1000 + GLB.NodeID,
				CO_Index		:= 16#41C0,
				CO_SubIndex		:= 16#14,
				DataLength		:= 2,
				WriteData		:= WriteData,
				StartWriting	:= TRUE	
			);	
			Index := Index + 1;
		ELSE
			SDO_WRITE();
		END_IF
			
		
	18: 
		IF SDO_WRITE.WriteDataFinished THEN
			FB_SDO_WRITE_REAL(	
				AdsNetID		:= GLB.ADSNetID_CAN,
				PortNr			:= 16#1000 + GLB.NodeID,
				CO_Index		:= 16#41C0,
				CO_SubIndex		:= 16#15,
				WriteData		:= Label.Rotor_inertia,
				StartWriting	:= TRUE	
			);	
			Index := Index + 1;
		ELSE
			SDO_WRITE();
		END_IF
			
		
	19: 
		IF FB_SDO_WRITE_REAL.WriteDataFinished THEN		
			FB_SDO_WRITE_REAL(	
				AdsNetID		:= GLB.ADSNetID_CAN,
				PortNr			:= 16#1000 + GLB.NodeID,
				CO_Index		:= 16#41C0,
				CO_SubIndex		:= 16#17,
				WriteData		:= Label.Motor_time_at_peak,
				StartWriting	:= TRUE	
			);	
			Index := Index + 1;
		ELSE
			FB_SDO_WRITE_REAL();
		END_IF
			
		
	20: 
		IF FB_SDO_WRITE_REAL.WriteDataFinished THEN		
			FB_SDO_WRITE_REAL(	
				AdsNetID		:= GLB.ADSNetID_CAN,
				PortNr			:= 16#1000 + GLB.NodeID,
				CO_Index		:= 16#41C0,
				CO_SubIndex		:= 16#18,
				WriteData		:= Label.Drive_time_at_peak,
				StartWriting	:= TRUE	
			);	
			Index := Index + 1;
		ELSE
			FB_SDO_WRITE_REAL();
		END_IF
			
		
	21: 
		IF FB_SDO_WRITE_REAL.WriteDataFinished THEN
			WriteData[0] := Label.Singleturn_resolution;
			WriteData[1] := 0;
			WriteData[2] := 0;
			WriteData[3] := 0;			
			SDO_WRITE(	
				AdsNetID		:= GLB.ADSNetID_CAN,
				PortNr			:= 16#1000 + GLB.NodeID,
				CO_Index		:= 16#41C0,
				CO_SubIndex		:= 16#19,
				DataLength		:= 1,
				WriteData		:= WriteData,
				StartWriting	:= TRUE	
			);	
			Index := Index + 1;
		ELSE
			FB_SDO_WRITE_REAL();
		END_IF
			
		
	22: 
		IF SDO_WRITE.WriteDataFinished THEN
			WriteData[0] := Label.Multiturn_resolution;
			WriteData[1] := 0;
			WriteData[2] := 0;
			WriteData[3] := 0;		
			SDO_WRITE(	
				AdsNetID		:= GLB.ADSNetID_CAN,
				PortNr			:= 16#1000 + GLB.NodeID,
				CO_Index		:= 16#41C0,
				CO_SubIndex		:= 16#1A,
				DataLength		:= 1,
				WriteData		:= WriteData,
				StartWriting	:= TRUE	
			);	
			Index := Index + 1;
		ELSE
			SDO_WRITE();
		END_IF
		
	
	23: // SAVE
		IF SDO_WRITE.WriteDataFinished THEN
			WriteData[0] := 0;
			WriteData[1] := 0;
			WriteData[2] := 0;
			WriteData[3] := 0;		
			SDO_WRITE(	
				AdsNetID		:= GLB.ADSNetID_CAN,
				PortNr			:= 16#1000 + GLB.NodeID,
				CO_Index		:= 16#1010,
				CO_SubIndex		:= 16#4,
				DataLength		:= 4,
				WriteData		:= WriteData,
				StartWriting	:= TRUE	
			);	
			Index := Index + 1;
		ELSE
			SDO_WRITE();
		END_IF		
			
			
	24: // Wait 500 ms for save process
		fbTonDelay(IN := TRUE, PT:= T#500MS);
		IF fbTonDelay.Q THEN
			fbTonDelay(IN := FALSE);
			Index := Index + 1;	
		END_IF
		
		
	255: // Finished 
		Finished := TRUE;
			
		
	ELSE
		Index := 255;
	
END_CASE

END_FUNCTION_BLOCK
